(* CODESYS project tc2_mc2.library
   Company: Beckhoff Automation GmbH
   DefaultNamespace: Tc2_MC2
   Version: 3.3.54.0
   Placeholder: Tc2_MC2
   Author: Beckhoff Automation GmbH
   Description: TwinCAT Motion Control Library (PlcOpen) v2.0
   Title: Tc2_MC2

Project tree, tasks and I/O mapping:
  libraries: Tc2_Math, * (Beckhoff Automation GmbH); Tc2_Standard, * (Beckhoff Automation GmbH); Tc2_System, * (Beckhoff Automation GmbH); Tc3_Module, * (Beckhoff Automation GmbH)
  Data types/
    [Internal]/
      DriveOperationMode/
        data type _ST_TcNC_ReadDriveOperationModeRequest
        data type _ST_TcNC_ReadDriveOperationModeResponse
        data type _ST_TcNC_WriteDriveOperationMode
      TcNC/
        ADS Axis/
          data type _ST_NCADS_Axis
          data type _ST_NCADS_AxisFunctions
          data type _ST_NCADS_AxisParameter
          data type _ST_NCADS_AxisState
          data type _ST_NCADS_IDXOFFS_AxisFunctions
          data type _ST_NCADS_IDXOFFS_AxisParameter
          data type _ST_NCADS_IDXOFFS_AxisState
        ADS Table/
          data type _ST_NCADS_IDXOFFS_TableFunctions
          data type _ST_NCADS_IDXOFFS_TableParameter
          data type _ST_NCADS_Table
          data type _ST_NCADS_TableFunctions
          data type _ST_NCADS_TableParameter
        data type _E_TcNC_CmdState
        data type _E_TcNC_CmdTypeNewTargPosAndVelo
        data type _E_TcNC_PosSetType
        data type _E_TcNC_ServoState
        data type _E_TcNC_SlaveTypes
        data type _E_TcNC_StartPosType
        data type _E_TcNC_TargPosType
        data type _ST_TcNC_Compensation2
        data type _ST_TcNC_CoupleSlave
        data type _ST_TcNC_CoupleSlaveMultiMaster
        data type _ST_TcNC_CoupleSlaveMultiMaster2
        data type _ST_TcNC_DecoupleSlave
        data type _ST_TcNc_OperationModes
        data type _ST_TcNC_PhasingRequest
        data type _ST_TcNC_SetEncoderSaclingFactor
        data type _ST_TcNC_SetPos
        data type _ST_TcNC_SetPosOnTheFly
        data type _ST_TcNc_SinusMotion
        data type _ST_TcNC_StopInfoRequest
        data type _ST_TcNC_StopInfoResponse
        data type _ST_TcNc_TouchProbeActivation
        data type _ST_TcNc_TouchProbeDeactivation
        data type _ST_TcNc_TouchProbeStatusRequest
        data type _ST_TcNc_TouchProbeStatusResponse
        data type _ST_TcNC_UniversalAxisTorqueStartRequest
        data type _ST_TcNC_UnversalAxisStartRequest
        data type _ST_TcNC_UnversalAxisStartResponse
      data type _E_ParameterType
      data type _E_PhasingState
      data type _E_ReadWriteParameterMode
      data type _E_SinusMotionMode
      data type _E_TcMC_STATES
      data type _E_TouchProbeState
      data type _InternalAxisRefData
      data type _ST_FunctionBlockResults
      data type _ST_NcIoOutputData
      data type _ST_ParaStruct
    Axis Reference/
      function block AXIS_REF [ST]: ReadStatus
      data type ST_AdsAddress
    BacklashCompensation/
      data type ST_BacklashCompensationOptions
    DriveOperationMode/
      data type E_DriveOperationMode
      data type ST_DriveOperationModeOptions
    Gearing/
      data type E_GearInMultiMasterSyncMode
      data type ST_GearInDynOptions
      data type ST_GearInMultiMasterOptions
      data type ST_GearInOptions
      data type ST_GearOutOptions
    Homing/
      data type E_EncoderReferenceMode
      data type MC_HomingMode
      data type ST_HomingOptions
    Motion/
      data type E_JogMode
      data type E_PositionType
      data type MC_BufferMode
      data type MC_Direction
      data type ST_MoveOptions
    Nc Process Data/
      data type E_NcIoDevice
      data type E_NcIoOutput
    Phasing/
      data type E_PhasingType
      data type ST_PhasingOptions
    Position Correction/
      data type E_AxisPositionCorrectionMode
      data type ST_PositionCompensationOptions
      data type ST_PositionCompensationTableElement
      data type ST_PositionCompensationTableParameter
    SelectControlLoop/
      data type E_SelectControlLoopType
      data type ST_SelectControlLoop
    Status and Parameter/
      data type E_AxisErrorCodes
      data type E_DisableMode
      data type E_NcAxisType
      data type E_NcDriveType
      data type E_NcEncoderType
      data type E_ReadMode
      data type E_SetScalingFactorMode
      data type E_WorkDirection
      data type MC_AxisParameter
      data type MC_AxisStates
      data type ST_AxisComponents
      data type ST_AxisOpModes
      data type ST_AxisParameterSet
      data type ST_AxisStatus
      data type ST_DriveAddress
      data type ST_McOutputs
      data type ST_NcApplicationRequest
      data type ST_PowerOptions
      data type ST_SetEncoderScalingOptions
      data type ST_SetPositionOptions
      data type ST_TableCharacValues
    Stepper/
      data type E_DestallDetectMode
      data type E_DestallMode
      data type ST_PowerStepperStruct
    Superposition/
      data type E_SuperpositionAbortOption
      data type E_SuperpositionMode
      data type ST_SuperpositionOptions
    Torque Control/
      data type ST_TorqueControlOptions
    Touch Probe/
      data type E_SignalEdge
      data type E_SignalSource
      data type E_TouchProbe
      data type E_TouchProbeMode
      data type MC_TouchProbeRecordedData
      data type TRIGGER_REF
  Global Variables/
    global variables Global_Variables
  POUs/
    [Internal]/
      ADS/
        function block _TcMC_ADSRDWRT [ST]
        function block _TcMC_ADSREAD [ST]
        function block _TcMC_ADSWRITE [ST]
      Axis Status Flag Functions/
        function F_AxisCamDataQueued [ST]
        function F_AxisCamScalingPending [ST]
        function F_AxisCamTableQueued [ST]
        function F_AxisControlLoopClosed [ST]
        function F_AxisDriveLimitActive [ST]
        function F_AxisExternalLatchValid [ST]
        function F_AxisGotNewTargetPosition [ST]
        function F_AxisHasBeenStopped [ST]
        function F_AxisHasExtSetPointGen [ST]
        function F_AxisHasJob [ST]
        function F_AxisInErrorState [ST]
        function F_AxisInPositionWindow [ST]
        function F_AxisInProtectedMode [ST]
        function F_AxisInPTPmode [ST]
        function F_AxisIoDataIsInvalid [ST]
        function F_AxisIsAtTargetPosition [ST]
        function F_AxisIsCalibrated [ST]
        function F_AxisIsCalibrating [ST]
        function F_AxisIsCompensating [ST]
        function F_AxisIsCoupled [FBD]
        function F_AxisIsMoving [ST]
        function F_AxisIsMovingBackwards [ST]
        function F_AxisIsMovingEndless [ST]
        function F_AxisIsMovingForward [ST]
        function F_AxisIsNotMoving [ST]
        function F_AxisIsReady [ST]
        function F_AxisJobPending [ST]
        function F_AxisMotionCommandsLocked [ST]
        function F_AxisPhasingActive [ST]
        function F_AxisReachedConstantVelocity [ST]
      Beta Function Blocks/
        Position Correction/
          function block MC_TableBasedPositionCompensation [ST]
        Sinus motion/
          function block MC_SinusOscillation [ST]
          function block MC_SinusSequence [ST]
        function block MC_ReadApplicationRequest [ST]
        function block MC_ReadStopInfo [ST]
      Objects/
        data type _FBAXIS_REF
        function block _TCMCGLOBAL [ST]: ReadDeviceInfo
      function _F_AxisState [ST]
      function _F_GetIndexGroup [ST]
      function _F_GetTcAxisObjectId [ST]
      function _F_GetTcDriveObjectId [ST]
      function _F_GetTcEncoderObjectId [ST]
      function _F_Init [ST]
      function _F_NcCycleCounterUpdated [ST]
      function _F_NcNoOfCycleCounterUpdated [ST]
      function _F_ReadStatus [ST]
      function _F_TcMC_DWORD_TO_HEXSTR [ST]
      function _F_TcMC_DWORD_TO_HEXSTR2 [ST]
      function _F_TcMC_IsValidAxisRef [ST]
      function _F_TcMC_IsValidRef [ST]
      function _F_TcMC_Round [ST]
      function _F_UpdateNcCycleCounter [ST]
      function block _FB_MoveSinusGeneric [ST]
      function block _FB_MoveUniversalGeneric [ST]: ActCalcDiffCmdNo, ActErrorMessage, ActMonitorAbortTorque, ActMonitorContinousMotion, ActMonitorContinuousTorque, ActMonitorDiscreteMotion, ActMonitorStop, ActNcCycleCounter
      function block _FB_PhasingGeneric [ST]
      function block _FB_PositionCorrectionTableLookup [ST]: ActIsCompensationDirection
      function block _FB_ReadWriteParameter [ST]
      function block _FB_WriteParameterPersistent [ST]
    [obsolete]/
      function F_GetVersion_TcMC2 [ST]
    Administrative/
      Axis Functions/
        function block MC_Power [ST]
        function block MC_Reset [ST]
        function block MC_SetPosition [ST]
      Extensions/
        DriveOperationMode/
          function block MC_ReadDriveOperationMode [ST]
          function block MC_WriteDriveOperationMode [ST]
        function block MC_BacklashCompensation [ST]
        function block MC_CalcDynamicsByRampTime [ST]
        function block MC_OverrideFilter [ST]
        function block MC_PositionCorrectionLimiter [ST]
        function block MC_PowerStepper [ST]
        function block MC_ReadDriveAddress [ST]
        function block MC_SelectControlLoop [ST]
        function MC_SetAcceptBlockedDriveSignal [ST]
        function block MC_SetEncoderScalingFactor [ST]
        function block MC_SetOverride [ST]
        function block MC_WriteNcIoOutput [ST]
      External Set Point Generator/
        function block MC_ExtSetPointGenDisable [ST]
        function block MC_ExtSetPointGenEnable [ST]
        function MC_ExtSetPointGenFeed [ST]
      Status and Parameter/
        function block MC_ReadActualPosition [ST]
        function block MC_ReadActualVelocity [ST]
        function block MC_ReadAxisComponents [ST]
        function block MC_ReadAxisError [ST]
        function block MC_ReadBoolParameter [ST]
        function block MC_ReadLargeParameter [ST]
        function block MC_ReadParameter [ST]
        function block MC_ReadParameterSet [ST]: ActGetSizeOfParameterSet
        function block MC_ReadStatus [ST]
        function block MC_WriteBoolParameter [ST]
        function block MC_WriteBoolParameterPersistent [ST]
        function block MC_WriteLargeParameter [ST]
        function block MC_WriteLargeParameterPersistent [ST]
        function block MC_WriteParameter [ST]
        function block MC_WriteParameterPersistent [ST]
      Touch Probe/
        function block MC_AbortTrigger [ST]
        function block MC_TouchProbe [ST]: ActTouchProbeActivate, ActTouchProbeMonitorActivity, ActTouchProbeMonitoring, ActTouchProbeMonitorLatchValid, ActTouchProbeMonitorPlcEvent, ActTouchProbeStartupInit
    Motion/
      Gearing/
        function block MC_GearIn [ST]: ActGearInDyn, WriteGearRatio
        function block MC_GearInDyn [ST]
        function block MC_GearInMultiMaster [ST]: ActGearInMultiMasterV1, ActGearInMultiMasterV2
        function block MC_GearOut [ST]
      Homing/
        function block MC_Home [ST]
      Manual Motion/
        function block MC_Jog [ST]: ActCheckJogEnd, ActJogMove
      Phasing/
        function block MC_HaltPhasing [FBD]
        function block MC_PhasingAbsolute [FBD]
        function block MC_PhasingRelative [FBD]
      Point To Point Motion/
        function block MC_Halt [FBD]
        function block MC_MoveAbsolute [FBD]
        function block MC_MoveAdditive [FBD]
        function block MC_MoveContinuousAbsolute [FBD]
        function block MC_MoveContinuousRelative [FBD]
        function block MC_MoveModulo [ST]: MC_MoveModuloCall
        function block MC_MoveRelative [FBD]
        function block MC_MoveVelocity [FBD]
        function block MC_Stop [ST]: ActStop
      Superposition/
        function block MC_AbortSuperposition [ST]
        function block MC_MoveSuperImposed [ST]
      Torque Control/
        function block MC_AbortTorqueControl [FBD]
        function block MC_TorqueControl [FBD]
  Version/
    global variables Global_Version
*)

// Data types/[Internal]/DriveOperationMode/_ST_TcNC_ReadDriveOperationModeRequest
{attribute 'conditionalshow'}
TYPE _ST_TcNC_ReadDriveOperationModeRequest :
STRUCT
	nReserved1 : UDINT;	// RESERVED1 (e.g. 'ULONG nCtrlLoopIndex')
	nReserved2 : UDINT;	// TC3 specific (natural alignment)
END_STRUCT
END_TYPE

// Data types/[Internal]/DriveOperationMode/_ST_TcNC_ReadDriveOperationModeResponse
{attribute 'conditionalshow'}
TYPE _ST_TcNC_ReadDriveOperationModeResponse :
STRUCT
	eTcNc3DrvOpMode : E_DriveOperationMode;	// >=0 [1] actual drive operation mode (enum NC3 Drive Operation Modes) (NC data type equal to ULONG)
    nReserved		: UDINT;	// RESERVED (e.g. OTCID    nObjectId, data type OTCID is equal to ULONG)
END_STRUCT
END_TYPE

// Data types/[Internal]/DriveOperationMode/_ST_TcNC_WriteDriveOperationMode
{attribute 'conditionalshow'}
TYPE _ST_TcNC_WriteDriveOperationMode :
STRUCT
	eTcNc3DrvOpMode : E_DriveOperationMode;	// enum NC3 Drive Operation Modes (signed value)(NC data type equal to ULONG)
	nReserved0 : UDINT;	// RESERVED1 (e.g. ULONG nCtrlLoopIdx [0;1,2,...])
	nReserved1 : UDINT; // RESERVED2 (e.g. 'OTCID nObjectId', data type equal to ULONG) (ObjId 0x0 is invalid, ObjID 0xFFFFFFFF is a joker (always allowed))
	nReserved2 : UDINT; // RESERVED3 
END_STRUCT
END_TYPE

// Data types/[Internal]/TcNC/ADS Axis/_ST_NCADS_Axis
{attribute 'conditionalshow'}
TYPE _ST_NCADS_Axis :
STRUCT
	Parameter	:	_ST_NCADS_AxisParameter;
	State		:	_ST_NCADS_AxisState;
	Functions	:	_ST_NCADS_AxisFunctions;
END_STRUCT
END_TYPE

// Data types/[Internal]/TcNC/ADS Axis/_ST_NCADS_AxisFunctions
{attribute 'conditionalshow'}
TYPE _ST_NCADS_AxisFunctions :
STRUCT
	IDXGRP		:	UDINT := 16#4200;
	IDXOFFS	:	_ST_NCADS_IDXOFFS_AxisFunctions;
END_STRUCT
END_TYPE

// Data types/[Internal]/TcNC/ADS Axis/_ST_NCADS_AxisParameter
{attribute 'conditionalshow'}
TYPE _ST_NCADS_AxisParameter :
STRUCT
	IDXGRP		:	UDINT := 16#4000;
	IDXOFFS	:	_ST_NCADS_IDXOFFS_AxisParameter;
END_STRUCT
END_TYPE

// Data types/[Internal]/TcNC/ADS Axis/_ST_NCADS_AxisState
{attribute 'conditionalshow'}
TYPE _ST_NCADS_AxisState :
STRUCT
	IDXGRP		:	UDINT := 16#4100;
	IDXOFFS	:	_ST_NCADS_IDXOFFS_AxisState;
END_STRUCT
END_TYPE

// Data types/[Internal]/TcNC/ADS Axis/_ST_NCADS_IDXOFFS_AxisFunctions
{attribute 'conditionalshow'}
TYPE _ST_NCADS_IDXOFFS_AxisFunctions :
STRUCT
	RESET					: UDINT := 16#0001;
	STOP					: UDINT := 16#0002;
	CLEAR					: UDINT := 16#0003;
	EMERGENCYSTOP		: UDINT := 16#0004;
	PARAMETRIZEDSTOP	: UDINT := 16#0005;
	INITIALIZE				: UDINT := 16#0007;	(* Initialize Axis *)
	ORIENTEDSTOP			: UDINT := 16#0009;	(* 19.04.04 issue #2470 *)
	CALIBR					: UDINT := 16#0010;
	NEWTARGPOS			: UDINT := 16#0011;
	NEWTARGPOSANDVELO	: UDINT := 16#0012;
	CHANGEDYNAMICPARAM	: UDINT := 16#0015;	(* NEU: Neue Dynamikparameter (Acc;Dec) fuer Positionierung *)
	UNIVERSALSTART		: UDINT := 16#0016;	(* 05.03.07: new 'axis start and restart' command with buffer mode (issue #2786+#3276) *)
	SLAVEUNIVERSALSTART	: UDINT := 16#0017;	(* 24.02.09: decoupling command with succeding universal axis start commanded to a slave axis *)
	RELEASEAXISLOCK			: UDINT := 16#0018; (* 10.12.18 release axis lock for motion commands *)
(*	ONLINESTART			: UDINT := 16#0017;*)	(* 05.03.07: new 'axis start and restart' command (online start) (issue #2786+#3276) *)
	SETEXTERNALERROR	: UDINT := 16#0019;	(* 06.10.04: Externen Achsfehler setzen (Laufzeitfehler) issue #2665 *)
	SETPOS					: UDINT := 16#001A;
	SETCALFLAG			: UDINT := 16#001B;	(* "ist referenziert"-Flag setzen *)
	SETACTPOS				: UDINT := 16#001C;	(* nur Istwertsetzen ohne Sollwertaenderung !!! *)
	SETDRIVEPOS			: UDINT := 16#001D;	(* antriebsseitiges Istwertsetzen *)
	SETENCODERSCALING	: UDINT := 16#001E;	(* 17.07.08: "Fliegende Änderung des Skalierungsfaktors" *)
	SETPOSONTHEFLY		: UDINT := 16#001F;	(* 29.11.05: "Fliegendes Istwert Setzen" (betrifft Ist - und Sollwert) (issue #3017) *)
	START					: UDINT := 16#0020;
	STARTEXT				: UDINT := 16#0021;
	STARTVELOCHANGE		: UDINT := 16#0022;	(* special function for MMW *)
	ENABLEEXTGEN			: UDINT := 16#0023;	(* enable/start external setpoint values *)
	DISABLEEXTGEN			: UDINT := 16#0024;	(* disable/stop external setpoint values *)
	REVERSINGSEQUENCE	: UDINT := 16#0025;
	STARTDRVOUT			: UDINT := 16#0026;
	STOPDRVOUT			: UDINT := 16#0027;
	CHANGEDRVOUT		: UDINT := 16#0028;
	JUMPTOOVERRIDE		: UDINT := 16#0029;	(* 04.11.04: jump to actual override value and froze them until change (issue #2697) *)
(*	SETABSOLUTEMEASURING: UDINT := 16#002A;	removed 20091106 KSt *)	(* 29.11.05: "Fliegendes Istwert Setzen" (betrifft Ist - und Sollwert) (issue #3017) *)
	EXTSETGENUNIVERSALSTART	: UDINT := 16#002B;	(* 23.11.10: deactivation of external setpoint generator with succeding universal axis start command *)
	UNIVERSALTORQUESTART	: UDINT := 16#002D;	(* 20181210 Fap -  new 'axis torque control start and restart' command with buffer mode *)
	STARTSCOM			: UDINT := 16#0030;	(* start superposition (position compensation) - 21.12.04: nun auch als 'ReadWrite'-Kommando *)
	STOPSCOM				: UDINT := 16#0031;	(* stop superposition (position compensation) *)
	PHASINGREQEUST		: UDINT := 16#0034;	(* start/stop the additional phasing set point generator used for a master/slave phase shift *)
	CPL						: UDINT := 16#0040;	(* Achse koppeln *)
	DECPL					: UDINT := 16#0041;	(* Achse entkoppeln (und optional neue Endposition mit neuer Geschwindigkeit) *)
	CPLCHANGE				: UDINT := 16#0042;	(* Achse Koppelparams ändern *)
	TABCPLCHANGE			: UDINT := 16#0043;	(* 3x TabSlaveAxe Tabelle-Koppelparams ändern *)
	STOPSLAVE				: UDINT := 16#0044;	(* Slave-Stop (Diagonal-Slave / Flying Saw) *)
	CPLTAB					: UDINT := 16#0045;	(* TabSlaveAxe Koppelparams setzen *)
	TABSLVACTIVCOR		: UDINT := 16#0046;	(* 2x TabSlaveAxe Korrekturtabelle aktivieren (mit/ohne Aktivierungsposition) *)
	TABSLVLEAVECYC		: UDINT := 16#0047;	(* TabSlaveAxe	Monozyklische Tabelle beenden *)
	TABSLVCOROFFSET		: UDINT := 16#0048;	(* TabSlaveAxe	Letzter Korrektur Offset *)
	TABSLVSCALING			: UDINT := 16#0049;	(* NEU: Slave-Skalierung der Solo-Tabellenkopplung setzen *)
	CPLSOLOTAB			: UDINT := 16#004A;	(* Solo Tabellen Kopplung *)
	CPLSYNCHRONIZING		: UDINT := 16#004B;	(* Slave Synchronizing Generator ('GearInPos' and 'GearInVelo') *)
	CAMSCALING			: UDINT := 16#004D;	(* Slave Change CAM Scaling (Aenderung der Tabellenskalierung) (issue #2514) *)
	DISABLE				: UDINT := 16#0050;	(* Achse sperren *)
	ENABLE					: UDINT := 16#0051;	(* Achse reaktivieren *)
	CHANGEAXISCTRLLOOP	: UDINT := 16#0052;	(* NEU: Aenderung des aktiven Achsregelkreises *)
	DRIVEDISABLE			: UDINT := 16#0060;	(* Drive-Output der Achse sperren *)
	DRIVEENABLE			: UDINT := 16#0061;	(* Drive-Output der Achse reaktivieren *)
	RELEASEBRAKE			: UDINT := 16#0062;	(* Feststellbremse loesen (Eil/Schleich-Gruppe) *)
	RECONFIGURATE		: UDINT := 16#0070;	(* Achse zurueckfuehren in eigene PTP-Gruppe *)
END_STRUCT
END_TYPE

// Data types/[Internal]/TcNC/ADS Axis/_ST_NCADS_IDXOFFS_AxisParameter
{attribute 'conditionalshow'}
TYPE _ST_NCADS_IDXOFFS_AxisParameter :
STRUCT
	(* NC ADS Index Offsets for Axis Parameters *)
	PARAMSTRUCT				: UDINT := 16#0000;
	ID							: UDINT := 16#0001;
	NAME						: UDINT := 16#0002;
	AXISTYPE					: UDINT := 16#0003;
	CYCLETIME					: UDINT := 16#0004;
	UNITNAME					: UDINT := 16#0005;
	VELOREFSEARCH			: UDINT := 16#0006;
	VELOSYNCSEARCH			: UDINT := 16#0007;
	VELOSLOWMANUAL			: UDINT := 16#0008;
	VELOFASTMANUAL			: UDINT := 16#0009;
	VELOFAST					: UDINT := 16#000A;
	POSAREAENABLE			: UDINT := 16#000F;
	POSAREARANGE			: UDINT := 16#0010;
	MOTCNTRLENABLE			: UDINT := 16#0011;
	MOTCNTRLTIME				: UDINT := 16#0012;
	LOOPENABLE				: UDINT := 16#0013;
	LOOPDISTANCE				: UDINT := 16#0014;
	TARGETPOSENA			: UDINT := 16#0015;
	TARGETPOSRANGE			: UDINT := 16#0016;
	TARGETPOSTIME			: UDINT := 16#0017;
	PULSDISTPOS				: UDINT := 16#0018;
	PULSDISTNEG				: UDINT := 16#0019;
	FADINGACCELERATION		: UDINT := 16#001D;
	FASTAXISSTOPSIGNALTYPE	: UDINT := 16#001E;
	UNITFLAGS					: UDINT := 16#0026;
	VELOMAXIMUM				: UDINT := 16#0027;
	MOTCNTRLRANGE			: UDINT := 16#0028;
	PEHCONTROLENA			: UDINT := 16#0029;
	PEHCONTROLTIME			: UDINT := 16#002A;
	BACKLASHCOMPENA			: UDINT := 16#002B;
	BACKLASH					: UDINT := 16#002C;
	DATAPERSISTENCE			: UDINT := 16#0030;
	HWAMSADDR				: UDINT := 16#0031;
	HWCHNNO					: UDINT := 16#0032;
	APPLICATIONREQUEST 		: UDINT := 16#0033;
	ACC							: UDINT := 16#0101;
	DEC						: UDINT := 16#0102;
	JERK						: UDINT := 16#0103;
	DELAY						: UDINT := 16#0104;
	OVERRIDETYPE				: UDINT := 16#0105;
	VELOJUMPFACTOR			: UDINT := 16#0106;
	REDUCTIONFEEDBACK		: UDINT := 16#0107;
	TOLERANCEBALLAUXAXIS	: UDINT := 16#0108;
	MAXPOSDEVIATIONAUXAXIS 	: UDINT := 16#0109;
	FASTACC					: UDINT := 16#010A;
	FASTDEC					: UDINT := 16#010B;
	FASTJERK					: UDINT := 16#010C;
	REF_POS						: UDINT := 16#0001_0103;
	ENCSEARCHDIR				: UDINT := 16#0001_0101;
	ENCSYNCDIR					: UDINT := 16#0001_0102;
	ENCREFMODE					: UDINT := 16#0001_0107;

(*
	SCALE						= TCNC_IDXOFFS_AXmappedENC | 0x00000006;	// 0x00010006;
	ENABLESOFTENDMIN		= TCNC_IDXOFFS_AXmappedENC | 0x0000000B;	// 0x0001000B;
	ENABLESOFTENDMAX		= TCNC_IDXOFFS_AXmappedENC | 0x0000000C;	// 0x0001000C;
	SOFTENDMIN				= TCNC_IDXOFFS_AXmappedENC | 0x0000000D;	// 0x0001000D;
	SOFTENDMAX				= TCNC_IDXOFFS_AXmappedENC | 0x0000000E;	// 0x0001000E;
	ENABLEPOSDIFF				= TCNC_IDXOFFS_AXmappedCTR | 0x00000010;	// 0x00020010;
	POSDIFFMAX				= TCNC_IDXOFFS_AXmappedCTR | 0x00000012;	// 0x00020012;
	GAINPOS					= TCNC_IDXOFFS_AXmappedCTR | 0x00000102;	// 0x00020102;
	VELOREF					= TCNC_IDXOFFS_AXmappedDRV | 0x00000101;	// 0x00030101;
*)
END_STRUCT
END_TYPE

// Data types/[Internal]/TcNC/ADS Axis/_ST_NCADS_IDXOFFS_AxisState
{attribute 'conditionalshow'}
TYPE _ST_NCADS_IDXOFFS_AxisState :
STRUCT
	ONLINESTRUCT					: UDINT := 16#0000;
	ERROR							: UDINT := 16#0001;
(*
	ACTPOS							= TCNC_IDXOFFS_AXmappedENC | 0x00000002;	// 0x00010002;
	ACTVELO						= TCNC_IDXOFFS_AXmappedENC | 0x00000005;	// 0x00010005;
	ACTACC							= TCNC_IDXOFFS_AXmappedENC | 0x00000006;	// 0x00010006;
	MODULOACTPOS				= TCNC_IDXOFFS_AXmappedENC | 0x00000003;	// 0x00010003;
	MODULOACTTURNS				= TCNC_IDXOFFS_AXmappedENC | 0x00000004;	// 0x00010004;
	ACTINCREMENTS				= TCNC_IDXOFFS_AXmappedENC | 0x00000007;	// 0x00010007;
*)
	SETTASKCYCLE					: UDINT := 16#0009;
	SETPOS							: UDINT := 16#000A;
	SETVELO						: UDINT := 16#000E;
	SETACC							: UDINT := 16#000F;
	MODULOSETPOS				: UDINT := 16#000B;
	MODULOSETTURNS				: UDINT := 16#000C;
	SETDIR							: UDINT := 16#000D;
	TARGETPOSITION				: UDINT := 16#0013;
	REMAININGTIMEANDPOS			: UDINT := 16#0014;
	STOPINFORMATION				: UDINT := 16#0018;
	SETTASKCYCLE_WITHOUTCORR	: UDINT := 16#0019;
	SETPOS_WITHOUTCORR			: UDINT := 16#001A;
	SETVELO_WITHOUTCORR		: UDINT := 16#001E;
	SETACC_WITHOUTCORR			: UDINT := 16#001F;
	SETDIR_WITHOUTCORR			: UDINT := 16#001D;
	COUPLESTATE					: UDINT := 16#0020;
	CPLPARAMS						: UDINT := 16#0022;
	CPLFACTOR						: UDINT := 16#0023;
	AXISCTRLLOOPIDX				: UDINT := 16#0024;
	AXISSETPOINTGENIDX			: UDINT := 16#0025;
	CPLCHARACVALUES				: UDINT := 16#0026;
	CAMINFO						: UDINT := 16#0027;
	CAMSTATUS					: UDINT := 16#0028;	(* activation status etc. *)
(*
	POSDIFF						= TCNC_IDXOFFS_AXmappedCTR | 0x0000000F;	// 0x0002000F;
*)
END_STRUCT
END_TYPE

// Data types/[Internal]/TcNC/ADS Table/_ST_NCADS_IDXOFFS_TableFunctions
{attribute 'conditionalshow'}
TYPE _ST_NCADS_IDXOFFS_TableFunctions :
STRUCT
	(* Index Offset definitions of table functions *)
	CREATETAB				: UDINT := 	16#0001_0000;		(* create table*)
	CREATEMOTIONTAB 		: UDINT := 	16#0001_0010;		(* create motion function table*)
	DELETETAB 				: UDINT := 	16#0002_0000; 		(* delete tables *)
END_STRUCT
END_TYPE

// Data types/[Internal]/TcNC/ADS Table/_ST_NCADS_IDXOFFS_TableParameter
{attribute 'conditionalshow'}
TYPE _ST_NCADS_IDXOFFS_TableParameter :
STRUCT
	MFREADCHARACVALUES	: UDINT := 	16#0000_0050;		(* read characteristic values of a motion function *)
	WRITETABROWS 		: UDINT := 	16#0100_0000;		(* write table *)
(*	WRITETABCOLS 			: UDINT := 	16#0200_0000;	*)	(* write table *)
	WRITEMFTABROWS 		: UDINT := 	16#0500_0000;		(* write motion function table *)
(*	WRITEMFTABCOLS 		: UDINT := 	16#0600_0000;	*)	(* write motion function table *)
(*	READSLAVEPOS 		: UDINT := 	16#0000_0021;	*)	(* read slave table position related to a master position *)
	MFREADTAB 			: UDINT := 	16#0000_0022;		(* read motion function as data table *)
	READSLAVEDYNAMICS 	: UDINT := 	16#0000_0023;		(* read slave table position, velocity and acceleration related to a master position *)
	READMASTERPOSITION 	: UDINT := 	16#0000_0024;		(* read master table position related  to slave position *)
END_STRUCT
END_TYPE

// Data types/[Internal]/TcNC/ADS Table/_ST_NCADS_Table
{attribute 'conditionalshow'}
TYPE _ST_NCADS_Table :
STRUCT
	Parameter	:	_ST_NCADS_TableParameter;
	Functions	:	_ST_NCADS_TableFunctions;
END_STRUCT
END_TYPE

// Data types/[Internal]/TcNC/ADS Table/_ST_NCADS_TableFunctions
{attribute 'conditionalshow'}
TYPE _ST_NCADS_TableFunctions :
STRUCT
	IDXGRP		:	UDINT := 16#A200;
	IDXOFFS	:	_ST_NCADS_IDXOFFS_TableFunctions;
END_STRUCT
END_TYPE

// Data types/[Internal]/TcNC/ADS Table/_ST_NCADS_TableParameter
{attribute 'conditionalshow'}
TYPE _ST_NCADS_TableParameter :
STRUCT
	IDXGRP		:	UDINT := 16#A000;
	IDXOFFS	:	_ST_NCADS_IDXOFFS_TableParameter;
END_STRUCT
END_TYPE

// Data types/[Internal]/TcNC/_E_TcNC_CmdState
{attribute 'conditionalshow'}
TYPE _E_TcNC_CmdState :
 (
	CMDSTATE_SUCCESSFULLY_EXECUTED				:= 1,	(* bit number *)
	CMDSTATE_ABORTED_WITHOUT_ERROR				:= 2,
	CMDSTATE_ENDED_WITH_ERROR					:= 3,
	CMDSTATE_LASTCMD_SUCCESSFULLY_EXECUTED	:= 8,
	CMDSTATE_LASTCMD_ABORTED_WITHOUT_ERROR	:= 9,
	CMDSTATE_LASTCMD_ENDED_WITH_ERROR			:= 10
 );
END_TYPE

// Data types/[Internal]/TcNC/_E_TcNC_CmdTypeNewTargPosAndVelo
{attribute 'conditionalshow'}
TYPE _E_TcNC_CmdTypeNewTargPosAndVelo :
 (
	TCNC_CHANGE_POS						:=  1,		(*Position (instantan)*)
	TCNC_CHANGE_VELO,							(*Geschwindigkeit (instantan)*)
	TCNC_CHANGE_POSANDVELO,					(*Position und Geschwindigkeit (instantan)*)
	TCNC_CHANGE_POS_AT_SWITCHPOS		:=  9,		(*Position (Umschaltposition)*)
	TCNC_CHANGE_VELO_AT_SWITCHPOS,			(*Geschwindigkeit (Umschaltposition)*)
	TCNC_CHANGE_POSANDVELO_AT_SWITCHPOS,	(*Position und Geschwindigkeit (Umschaltposition)*)
	TCNC_REACH_VELO_AT_POS				:= 14		(*neue Geschwindigkeit wird an einer bestimmten Position erreicht *)
 );
END_TYPE

// Data types/[Internal]/TcNC/_E_TcNC_PosSetType
{attribute 'conditionalshow'}
TYPE _E_TcNC_PosSetType : (* mode is used with MC_SetPosition *)
(
	TCNC_POSSETTYPE_ABSOLUTE		:= 1,	(*Absolute position*)
	TCNC_POSSETTYPE_RELATIVE			(*Relative position*)
) UINT;
END_TYPE

// Data types/[Internal]/TcNC/_E_TcNC_ServoState
{attribute 'conditionalshow'}
TYPE _E_TcNC_ServoState :
 (
	TCNC_INACTIVE 	:= 0,
	TCNC_RUNNING,
	TCNC_OVERRIDE_ZERO,			(* axis is executing a job but override is zero *)
	TCNC_PHASE_VELOCONST,		(* aixs is moving at constant velocity *)
	TCNC_PHASE_ACCPOS,			(* axis is accelerating *)
	TCNC_PHASE_ACCNEG,			(* axis is decelerating *)
	TCNC_PHASE_TORQUECONST,		(* 20181210 Fap - axis is moving at constant torque *)

	(* slaves only *)
	TCNC_PHASE_PREPHASE := 11, 	(* slave axis is in a motion pre-phase - slaves only *)
	TCNC_PHASE_SYNCHRONIZING, 	(* slave axis is synchronizzing slaves only *)
	TCNC_PHASE_SYNCHRONOUS, 	(* slaves only *)

	(* two speed axes only *)
	TCNC_PHASE_TWOSPEED_MOVING := 21,	(* GVGSTATE_TWOSPEED_21 *)

	(* external set point generation - from Tc 2.11 R2 *)
	TCNC_PHASE_EXTSETGEN_MODE1 := 41,	(* external set point generator active *)
	TCNC_PHASE_EXTSETGEN_MODE2		(* internal and external set point generator active *)
 );
END_TYPE

// Data types/[Internal]/TcNC/_E_TcNC_SlaveTypes
{attribute 'conditionalshow'}
TYPE _E_TcNC_SlaveTypes :
(
	TCNC_SLAVETYPE_LINEAR							:=	1,	(* Lineare Kopplung (Geradengleichung) *)
	TCNC_SLAVETYPE_FLYINGSAW_ONVELOCITY		:= 	2,	(* diagonal synchron. Aufkoppeln schnellstens auf Geschwindigkeit *)
	TCNC_SLAVETYPE_FLYINGSAW_ONPOSITION		:=	3,	(* diagonal synchron. Aufkoppeln auf Position und Geschwindigkeit *)
	TCNC_SLAVETYPE_FLYINGSAW_QUADRATIC		:=	4,	(* diagonal synchron. Aufkoppeln (quadratisches Geschw.-Profil) *)
	TCNC_SLAVETYPE_SYNCHRONIZING_ONVELO		:= 	5,	(* synchron. Aufkoppeln instantan auf Geschwindigkeit *)
	TCNC_SLAVETYPE_SYNCHRONIZING_ONPOS       	 	:= 	6,	(* synchron. Aufkoppeln auf Positionen und Geschwindigkeit *)
	TCNC_SLAVETYPE_SYNCJERKSETTER_ONVELO       	:= 	7,	(* synchron. Aufkoppeln auf Geschwindigkeit (zeitbasiert mittels Ruck-Steller) *)
	TCNC_SLAVETYPE_TABULAR						:=	10,	(* Tabellen-Kopplung ("simple/standard tabular slave") *)
	TCNC_SLAVETYPE_MULTITABULAR					:= 	11,	(* Tabellen-Kopplung ("multiscalable multi-tabular slave") *)
	TCNC_SLAVETYPE_FLYINGMODULO_LINEAR			:=	12,	(* Modulo Kopplung auf Position und/oder Geschwindigkeit mit anschliessender Linear Kopplung ("Schuette") *)
	TCNC_SLAVETYPE_MOTIONFUNCTIONTABULAR		:=	13,	(* Tabellen-Kopplung "motion functions" *)
	TCNC_SLAVETYPE_UNIVERSALTABULAR			:=	14,	(* Tabellen-Kopplung, universal tabular type substitues TABULAR, MULTITABULAR and MOTIONFUNCTION - 08.07.05 *)
	TCNC_SLAVETYPE_LINEAR_CYCLICCHANGES_RAMP	:=	15,	(* Lineare Kopplung (Geradengleichung) mit zyklischer Koppelfaktoraenderung *)
	TCNC_SLAVETYPE_BILINEAR						:=	16,	(* 27.04.01: Zweifach Lineare Kopplung (Geradengleichung)*)
	TCNC_SLAVETYPE_LINEAR_MULTIMASTER		:=	17,	(* 29.05.08: Lineare Multi-Master-Kopplung ('MC_GearInMultiMaster') *)
	TCNC_SLAVETYPE_CONST_SURFACEVELO_RAMP	:=	18	(* Verrechnete Winkelgeschwindigkeit fuer konstante Oberflaechengeschwindig. in Abhaengigkeit vom Radiusistwert des Enc.2 *)
);
END_TYPE

// Data types/[Internal]/TcNC/_E_TcNC_StartPosType
{attribute 'conditionalshow'}
TYPE _E_TcNC_StartPosType :
(
	TCNC_START_ABSOLUTE					:= 1,		(*Start to absolute position*)
	TCNC_START_RELATIVE					:= 2,		(*Start to relative position*)
	TCNC_START_ENDLESS_PLUS				:= 3,		(*Start to endless positive position*)
	TCNC_START_ENDLESS_MINUS			:= 4,		(*Start to endless negative position*)
	TCNC_START_MODULO					:= 5,		(*Start to modulo position *)
	TCNC_START_ADDITIVE					:= 6,		(*Start to a position relative to the last recent target position *)
	TCNC_START_MODULO_SHORT				:= 261, 	(*Start to modulo position *)
 	TCNC_START_MODULO_PLUS				:= 517, 	(*Start to modulo position *)
 	TCNC_START_MODULO_MINUS				:= 773, 	(*Start to modulo position *)
	TCNC_START_MODULO_CURRENT			:= 1029,	(* start to modulo position in current direction *)
 	TCNC_START_ABS_INTERNAL				:= 9, 		(*Start to absolute position, internal use*)
	TCNC_START_ENDLESSPLUS_SLOWMANUAL	:= 272,		(* manual jog mode *)
	TCNC_START_ENDLESSMINUS_SLOWMANUAL	:= 273,		(* manual jog mode *)
	TCNC_START_ENDLESSPLUS_FASTMANUAL	:= 528,		(* manual jog mode *)
	TCNC_START_ENDLESSMINUS_FASTMANUAL	:= 529,		(* manual jog mode *)
	TCNC_START_STOPANDLOCK				:= 4096,	(* stop axis and lock against any motion commands *)
	TCNC_START_HALT						:= 8192,	(* halt axis - can be interrupted by any motion commands *)
	TCNC_START_TORQUE_ABORT				:= 12288,	(* 20181210 Fap - halt torque control *)
	TCNC_START_TORQUE_ABSOLUTE			:= 12289,	(* 20181210 Fap - Start torque control absolute *)
	TCNC_START_TORQUE_RELATIVE			:= 12290	(* 20190108 Fap - Start torque control relative NOT IMPLEMENTED *)
) UINT;
END_TYPE

// Data types/[Internal]/TcNC/_E_TcNC_TargPosType
{attribute 'conditionalshow'}
TYPE _E_TcNC_TargPosType :
(
	TCNC_POS_ABSOLUTE		:= 1,	(*Absolute position*)
	TCNC_POS_RELATIVE,			(*Relative position*)
	TCNC_POS_MODULO			:= 5,	(*Modulo position*)
	TCNC_POS_ABS_INTERNAL	:= 9	(*Absolute position, internal use*)
);
END_TYPE

// Data types/[Internal]/TcNC/_ST_TcNC_Compensation2
{attribute 'conditionalshow'}
TYPE _ST_TcNC_Compensation2 :	(* internal use with MC_MoveSuperimposed_2 *)
STRUCT
	nCompType	:	UDINT;	(* E_SuperpositionMode *)
	nReserved1	:	UDINT;
	fAccPlus		:	LREAL;
	fAccMinus	:	LREAL;
	fVeloDiff		:	LREAL;
	fVeloProcess	:	LREAL;
	fDistance	:	LREAL;	(* distance to compensate *)
	fLength		:	LREAL;	(* distance moved during compensation *)
	nWarningId	: 	UDINT;	(* documented as error code *)
	nReserved2	:	UDINT;
END_STRUCT
END_TYPE

// Data types/[Internal]/TcNC/_ST_TcNC_CoupleSlave
{attribute 'conditionalshow'}
TYPE _ST_TcNC_CoupleSlave :
STRUCT
	nSlaveType		:	UDINT;
	nMasterAxisId	:	UDINT;
	nMasterSubIdx	:	UDINT;
	nSlaveSubIdx		:	UDINT;
	fCoupleParam1	:	LREAL;
	fCoupleParam2	:	LREAL;
	fCoupleParam3	:	LREAL;
	fCoupleParam4	:	LREAL;
END_STRUCT
END_TYPE

// Data types/[Internal]/TcNC/_ST_TcNC_CoupleSlaveMultiMaster
{attribute 'conditionalshow'}
TYPE _ST_TcNC_CoupleSlaveMultiMaster :
STRUCT
	nSlaveType		:	UDINT;
	nMasterAxisId	:	UDINT;
	nMasterSubIdx	:	UDINT;
	nSlaveSubIdx		:	UDINT;
(*	nMasterID1 = nMasterAxisId *)
	nMasterID2		:	UDINT;
	nMasterID3		:	UDINT;
	nMasterID4		:	UDINT;
	nMasterID5		:	UDINT;
	nMasterID6		:	UDINT;
	nMasterID7		:	UDINT;
	nMasterID8		:	UDINT;
	nReserved1		:	UDINT;
	fSlaveAcceleration:	LREAL;
	nCheckAndOpMode:	DWORD;
	nReserved2		:	UDINT;
END_STRUCT
END_TYPE

// Data types/[Internal]/TcNC/_ST_TcNC_CoupleSlaveMultiMaster2
{attribute 'conditionalshow'}
TYPE _ST_TcNC_CoupleSlaveMultiMaster2 :
STRUCT
	nSlaveType		:	UDINT;
	nMasterAxisId	:	UDINT;
	nMasterSubIdx	:	UDINT;
	nSlaveSubIdx		:	UDINT;
(*	nMasterID1 = nMasterAxisId *)
	nMasterID2		:	UDINT;
	nMasterID3		:	UDINT;
	nMasterID4		:	UDINT;
	nMasterID5		:	UDINT;
	nMasterID6		:	UDINT;
	nMasterID7		:	UDINT;
	nMasterID8		:	UDINT;
	nReserved1		:	UDINT;
	fSlaveMaxAcc	:	LREAL;
	nCheckAndOpMode : 	DWORD;
	nReserved2		:	UDINT;
(*	// Erweiterungen fuer NEW VERSION V2 *)
	fSlaveMaxDec	:	LREAL;
	fSlaveMaxJerk	:	LREAL;
	fSlaveMaxVelo	:	LREAL;
	fReserved3		:	LREAL;
	fReserved4		:	LREAL;
END_STRUCT
END_TYPE
(* 	nCheckAndOpMode is a 32 bit array
Bits:
 0:	VelocitySynchronizationOnly		
 1:	
 2:
*)

// Data types/[Internal]/TcNC/_ST_TcNC_DecoupleSlave
{attribute 'conditionalshow'}
TYPE _ST_TcNC_DecoupleSlave :
STRUCT
	nDecoupleMode	:	UDINT;
	nReserved		:	UDINT;
	fNewPosEnd	:	LREAL;
	fNewVeloRequ	:	LREAL;
	fAcceleration	:	LREAL;
	fDeceleration	:	LREAL;
	fJerk			:	LREAL;
END_STRUCT
END_TYPE

// Data types/[Internal]/TcNC/_ST_TcNc_OperationModes
{attribute 'conditionalshow'}
TYPE _ST_TcNc_OperationModes :
STRUCT
	(* OpModeDWord in cyclic interface *)
(*   0 *)	PosAreaControl	:	DWORD := 2#0000_0000_0000_0000_0000_0000_0000_0001;
(*   1 *)	TargetPosControl	:	DWORD := 2#0000_0000_0000_0000_0000_0000_0000_0010;
(*   2 *)(*	Loop			:	DWORD := 2#0000_0000_0000_0000_0000_0000_0000_0100;*)
(*   3 *)(*	MotionControl		:	DWORD := 2#0000_0000_0000_0000_0000_0000_0000_1000;*)
(*   4 *)(*	PEHTimeControl	:	DWORD := 2#0000_0000_0000_0000_0000_0000_0001_0000;*)
(*   5 *)(*	BacklashComp	:	DWORD := 2#0000_0000_0000_0000_0000_0000_0010_0000;*)
(*   6 *)(*	DelayedErrorReaction *)
(*   7 *)(*	Modulo *)
(*   8 *)(*	SimulationAxis *)
	(* bits 9 .. 11 reserved for supplement products *)
(*   12 *)	StopMonitoring 	:	DWORD := 2#0000_0000_0000_0000_0001_0000_0000_0000;
	(* bits 13 .. 15 reserved *)
(* 16 *)(*	PosDiffControl  	:	DWORD := 2#0000_0000_0000_0001_0000_0000_0000_0000;*)
(* 17 *)(*	VeloDiffControl	:	DWORD := 2#0000_0000_0000_0010_0000_0000_0000_0000;*)
(* 18 *)(*	SoftEndMinControl	:	DWORD := 2#0000_0000_0000_0100_0000_0000_0000_0000;*)
(* 19 *)(*	SoftEndMaxControl:	DWORD := 2#0000_0000_0000_1000_0000_0000_0000_0000;*)
(* 20 *)(*	ActPosCorrection	:	DWORD := 2#0000_0000_0001_0000_0000_0000_0000_0000;*)
(* 21 *)	AllowSlaveCommands :DWORD	:= 2#0000_0000_0010_0000_0000_0000_0000_0000;
(* 22 *)(*	AllowExtSetGenAxisCommands*)
(* 23 *)(*	ApplicationRequest*)
	(* bits 24 .. 31  *)
(* 24 *)(* 	NcStartTick : BYTE NC cycle counter *)
END_STRUCT
END_TYPE

// Data types/[Internal]/TcNC/_ST_TcNC_PhasingRequest
{attribute 'conditionalshow'}
TYPE _ST_TcNC_PhasingRequest :	(* internal use with MC_MoveSuperimposed_2 (NCADS_STARTPHASING) *)
STRUCT
	nPhasingType	:	UDINT;	(* phasing type absolute or relative *)
	nControlMask		:	UDINT;	(* internal control mask (RESERVED) *)
	nMasterAxisID	: 	UDINT;	(* Optional: master axis ID (for multi cam) *)
	nReserved1		: 	UDINT;

	fPhaseShift		:	LREAL;	(* phasing shift (distance)		[mm] *)
	fVelo			:	LREAL;	(* maximum velocity (> 0)		[mm/s] *)
	fAcc				:	LREAL;	(* maximum acceleration (>= 0)	[mm/s^2] *)
	fDec			:	LREAL;	(* maximum deceleration (>= 0)	[mm/s^2] *)
	fJerk			:	LREAL;	(* maximum jerk (>= 0)			[mm/s^3] *)

	fReserved		: 	ARRAY[2..5] OF LREAL;

	nReserved6		: 	UDINT;
	nBufferMode		: 	UDINT;	(* NOT USED YET: 'buffer mode' *)
	fBlendingPos		:	LREAL;	(* NOT USED YET: optional blending position *)
END_STRUCT
END_TYPE

// Data types/[Internal]/TcNC/_ST_TcNC_SetEncoderSaclingFactor
{attribute 'conditionalshow'}
TYPE _ST_TcNC_SetEncoderSaclingFactor :
STRUCT
 	nEncoderScalingFactorType	:	UINT;
	nCtrlWord					:	UINT; 	(* additional option flags *)	(* added KSt 2009-04-09 *)
	nReserved					:	UDINT;
	fEncoderScalingFactor		:	LREAL;
END_STRUCT
END_TYPE

// Data types/[Internal]/TcNC/_ST_TcNC_SetPos
{attribute 'conditionalshow'}
TYPE _ST_TcNC_SetPos :
STRUCT
	nPosIstType		:	UDINT;
	nReserved		:	UDINT;
	fNewPosIst		:	LREAL;
	fReserved		:	LREAL;
END_STRUCT
END_TYPE

// Data types/[Internal]/TcNC/_ST_TcNC_SetPosOnTheFly
{attribute 'conditionalshow'}
TYPE _ST_TcNC_SetPosOnTheFly :
STRUCT
	nPosSetType		: 	UDINT; 	(*_E_TcNC_PosSetType *)	(* Absolute, Relative - added KSt 2009-01-28 *)
	nCtrlDWord		:	UDINT; 	(* additional option flags *)	(* added KSt 2009-01-28 *)
 	fPreviousActualPos:	LREAL;	(* value not used any longer since 2009-01-28 *)
	fNewActualPos	:	LREAL;
	nReserved		:	ARRAY[1..2] OF DWORD;	(* added KSt 2009-01-28 *)
END_STRUCT
END_TYPE

// Data types/[Internal]/TcNC/_ST_TcNc_SinusMotion
{attribute 'conditionalshow'}
TYPE _ST_TcNc_SinusMotion :
STRUCT
	StartType 					: UDINT;
	BaseAmplitude 				: LREAL;
	BaseFrequency 				: LREAL;
	StartAmplitudeAtBeginn 		: LREAL;
	FeedConstantMotor 			: LREAL;
	StartFrequency 				: LREAL;
	StopFrequency 				: LREAL;
	StepDuration 				: LREAL;
	NumberMeasurements 			: UDINT;
	NumberParallelMeasurements 	: UDINT;
END_STRUCT
END_TYPE

// Data types/[Internal]/TcNC/_ST_TcNC_StopInfoRequest
{attribute 'conditionalshow'}
TYPE _ST_TcNC_StopInfoRequest :
STRUCT
	Deceleration : LREAL;
	Jerk	: LREAL;
END_STRUCT
END_TYPE

// Data types/[Internal]/TcNC/_ST_TcNC_StopInfoResponse
{attribute 'conditionalshow'}
TYPE _ST_TcNC_StopInfoResponse :
STRUCT
	StopDistance : LREAL;
	StopTime : LREAL;
END_STRUCT
END_TYPE

// Data types/[Internal]/TcNC/_ST_TcNc_TouchProbeActivation
{attribute 'conditionalshow'}
TYPE _ST_TcNc_TouchProbeActivation :
STRUCT
	TouchProbe 	: UDINT; 	(* number of probe unit 1..4 *)
	Edge		: UDINT; 	(* rising(0) or falling(1) signal edge *)
	Mode		: UDINT;	(* touch probe mode 0=single, 1=continuous *)
	SignalSource	: UDINT;	(* optional physical signal source used by the probe unit *)
	_reserved 	: ARRAY[1..2] OF UDINT;
END_STRUCT
END_TYPE

// Data types/[Internal]/TcNC/_ST_TcNc_TouchProbeDeactivation
{attribute 'conditionalshow'}
TYPE _ST_TcNc_TouchProbeDeactivation :
STRUCT
	TouchProbe 	: UDINT; 	(* number of probe unit 1..4 *)
	Edge		: UDINT; 	(* rising(0) or falling(1) signal edge *)
	_reserved 	: ARRAY[1..4] OF UDINT;
END_STRUCT
END_TYPE

// Data types/[Internal]/TcNC/_ST_TcNc_TouchProbeStatusRequest
{attribute 'conditionalshow'}
TYPE _ST_TcNc_TouchProbeStatusRequest :
STRUCT
	TouchProbe 	: UDINT; 	(* number of probe unit 1..4 *)
	_reserved 	: ARRAY[1..5] OF UDINT;
END_STRUCT
END_TYPE

// Data types/[Internal]/TcNC/_ST_TcNc_TouchProbeStatusResponse
{attribute 'conditionalshow'}
TYPE _ST_TcNc_TouchProbeStatusResponse :
STRUCT
	(* latch status data for the rising signal edge *)
	RisingEdgeActive 		: UDINT;
	RisingEdgeValid		: UDINT;
	RisingEdgeValue 		: LREAL;
	RisingEdgeCounter 	: UDINT;
	_reserved1 			: UDINT;

	(* latch status data for the falling signal edge *)
	FallingEdgeActive 	: UDINT;
	FallingEdgeValid		: UDINT;
	FallingEdgeValue 		: LREAL;
	FallingEdgeCounter	 : UDINT;
	_reserved2 			: UDINT;

	_reserved3 : ARRAY[1..4] OF UDINT;
END_STRUCT
END_TYPE

// Data types/[Internal]/TcNC/_ST_TcNC_UniversalAxisTorqueStartRequest
{attribute 'conditionalshow'}
TYPE _ST_TcNC_UniversalAxisTorqueStartRequest :
STRUCT
	nStartType			: UDINT;			(* axis start TYPE (TORQUECONTINUOUS) *)
	nControlMask		: UDINT;			(* optional: control mask *)

	nMode				: UDINT;			(* optional: mode (ENUM) *)
	nBufferMode			: UDINT;			(* 'buffer mode' OR 'activation mode' FOR 'buffered commands' (first Only ABORTING) *)

	fTorque				: LREAL;			(* target torque [signed]*)
	fTorqueRamp			: LREAL;			(* nc torque ramp *)

	fVelocityLimitHigh	: LREAL;			(* velocity limit high [signed]*)
	fVelocityLimitLow	: LREAL;			(* velocity limit low [signed]*)

	fAcceleration		: LREAL;			(* acceleration (>= 0) *)
	fDeceleration		: LREAL;			(* deceleration (>= 0) *)

	fManualTorque		: LREAL;			(* optional: manual torque (sync value) *)
END_STRUCT
END_TYPE

// Data types/[Internal]/TcNC/_ST_TcNC_UnversalAxisStartRequest
{attribute 'conditionalshow'}
TYPE _ST_TcNC_UnversalAxisStartRequest :
STRUCT
	nStartType	: UDINT;			(* axis start TYPE (ABSOLUT, RELATIV, ENDLESS_PLUS, ENDLESS_MINUS, MODULO_SHORT, MODULO_PLUS, MODULO_MINUS) *)
	nControlMask	: UDINT;			(* optional: control mask *)

	fPosTarget	: LREAL;			(* target position *)
	fVeloRequ	: LREAL;			(* required velocity *)

	fAcc			: LREAL;			(* acceleration (>= 0) *)
	fDec		: LREAL;			(* deceleration (>= 0) *)
	fJerk		: LREAL;			(* jerk (>= 0) *)

	nBufferMode	: UDINT;			(* optional: 'buffer mode' OR 'activation mode' FOR 'buffered commands' (issue #2786) *)
	nReserved	: UDINT;			(* reserved *)
	fBlendingPosition: LREAL;			(* optional: activation position *)

	fVeloStart	: LREAL;			(* optional: start velocity	(0 <= fVeloStart <= fVeloRequ)	Frage: erstmal weglassen ??? *)
	fVeloEnd		: LREAL;			(* optional: end velocity		(0 <= fVeloEnd <= fVeloRequ)	Frage: erstmal weglassen ??? *)
END_STRUCT
END_TYPE

// Data types/[Internal]/TcNC/_ST_TcNC_UnversalAxisStartResponse
{attribute 'conditionalshow'}
TYPE _ST_TcNC_UnversalAxisStartResponse :
STRUCT
	nCmdNo 	: WORD;			(* Continuous actual command number *)
	nCmdState	: WORD;			(* Command state *)
END_STRUCT
END_TYPE

// Data types/[Internal]/_E_ParameterType
{attribute 'conditionalshow'}
TYPE _E_ParameterType :
 (
	PARAMETERTYPE_NOTYPE := 0,
	PARAMETERTYPE_BOOL,
	PARAMETERTYPE_DWORD,
	PARAMETERTYPE_LREAL,
	PARAMETERTYPE_LARGE	// any parameter with size > LREAL; used for LINT or ULINT as well
 );
END_TYPE

// Data types/[Internal]/_E_PhasingState
{attribute 'conditionalshow'}
(* Phasing internal probe states *)
TYPE _E_PhasingState :
 (
	PhasingInactive,
	PhasingActivated,
	PhasingAborted
 );
END_TYPE

// Data types/[Internal]/_E_ReadWriteParameterMode
{attribute 'conditionalshow'}
TYPE _E_ReadWriteParameterMode :
 (
	READWRITEPARAMETERMODE_READ 	:=10,
	READWRITEPARAMETERMODE_WRITE	:= 11
 );
END_TYPE

// Data types/[Internal]/_E_SinusMotionMode
{attribute 'conditionalshow'}
TYPE _E_SinusMotionMode :
(
	eSinusMode_Oscillation := 0,
	eSinusMode_Sequence := 1	
);
END_TYPE

// Data types/[Internal]/_E_TcMC_STATES
{attribute 'conditionalshow'}
TYPE _E_TcMC_STATES :
 (
	STATE_INITIALIZATION  := 100,
	STATE_ORDER,
	STATE_RUNNING,
	STATE_WAITING,
	STATE_MOTIONCOMMANDSLOCKED
 );
END_TYPE

// Data types/[Internal]/_E_TouchProbeState
{attribute 'conditionalshow'}
(* MC_TouchProbe internal probe states *)
TYPE _E_TouchProbeState :
 (
	TouchProbeInactive,
	TouchProbeActivated,
	TouchProbeAborted
 );
END_TYPE

// Data types/[Internal]/_InternalAxisRefData
{attribute 'conditionalshow'}
TYPE _InternalAxisRefData :
STRUCT
	NcCycleCounterAvailable					: BOOL;	(* TRUE if the NcCycleCounter is definitely available on the target system - FALSE if undefined *)

	NcCycleCounter_AtReadStatusCall			: UDINT;	(* current NC cycle counter when calling ReadStatus *)
	LastTaskIndex_AtReadStatusCall 			: BYTE;	(* task index of last recent status update *)
	CounterSameTaskIndex_AtReadStatusCall 	: UINT;	(* counter increments to max 100 if the task index for the status update never changes *)

	PhasingState							: _E_PhasingState;	// KSt 20190703 global handshake for phasing blocks
END_STRUCT
END_TYPE

// Data types/[Internal]/_ST_FunctionBlockResults
{attribute 'conditionalshow'}
TYPE _ST_FunctionBlockResults :
STRUCT
	Done				:	BOOL;
	CommandAborted		:	BOOL;
	Error				:	BOOL;
{attribute 'displaymode':='hex'}
	ErrorID				:	UDINT;
{attribute 'displaymode':='dec'}
	BusyCounter			: 	UDINT; (* busy cycles since triggering the block - 2018-01-24 KSt *)
END_STRUCT
END_TYPE

// Data types/[Internal]/_ST_NcIoOutputData
{attribute 'conditionalshow'}
TYPE _ST_NcIoOutputData :
STRUCT
	ByteOffset				: UDINT;
	BitSelectMask			: UDINT;
	BitValues				: UDINT;
END_STRUCT
END_TYPE

// Data types/[Internal]/_ST_ParaStruct
{attribute 'conditionalshow'}
TYPE _ST_ParaStruct :
STRUCT
	Port		: 	UINT;	(* 2014-07-14 KSt *)
	IndexGroup 	:	UDINT;
	IndexOffset :	UDINT;
	ParaType	:	_E_ParameterType;
	LrealSize	:	UDINT; (* sizeof Lreal data array *)
	LrealOffset	: 	UDINT; (* offset in lreal data array *)
END_STRUCT
END_TYPE

// Data types/Axis Reference/ST_AdsAddress
TYPE ST_AdsAddress :
STRUCT
	NetId	 	: STRING(23);
	Port 		: UINT;
	Channel 	: UINT;
END_STRUCT
END_TYPE

// Data types/BacklashCompensation/ST_BacklashCompensationOptions
TYPE ST_BacklashCompensationOptions :
STRUCT
{attribute 'conditionalshow'}
	_reserved : BOOL;
END_STRUCT
END_TYPE

// Data types/DriveOperationMode/E_DriveOperationMode
TYPE E_DriveOperationMode :
(
	DriveOperationMode_Default						:= 0,   // 0x0000: default => reactivate the nc default op mode (if default mode is known!?!)
	// general operation modes (e.g. CANopen/CoE)
	DriveOperationMode_Torque   					:= 1,  	// 0x0001: torque control 
	DriveOperationMode_Velo1   						:= 2,	// 0x0002: velocity control with feedback 1
	DriveOperationMode_Velo2    					:= 3,   // 0x0003: velocity control with feedback 2
	DriveOperationMode_Pos1  		 	  			:= 4,   // 0x0004: pos control with feedback 1, lag less
	DriveOperationMode_Pos2     					:= 5,   // 0x0005: pos control with feedback 2, lag less
	DriveOperationMode_TorqueAndCommutationAngle	:= 6,   // 0x0006: torque control with commutation angle
	
	// new operation modes using dynamic container (also called 'dynamic MDT' or 'dynamic sync manager')
{attribute 'hide'}
	DriveOperationMode_TorqueDynContainer			:= 17,	// 0x0011: torque ctrl using dynamic container (READ ONLY !!!)
{attribute 'hide'}
	DriveOperationMode_Velo1DynContainer			:= 18,  // 0x0012: velo with ctrl feedback 1 using dynamic container (READ ONLY !!!)
{attribute 'hide'}
	DriveOperationMode_Velo2DynContainer			:= 19,  // 0x0013: velo with ctrl feedback 2 using dynamic container (READ ONLY !!!)
{attribute 'hide'}
	DriveOperationMode_Pos1DynContainer				:= 20,  // 0x0014: pos ctrl with feedback 1 (lag less) using dynamic container (READ ONLY !!!)
{attribute 'hide'}
	DriveOperationMode_Pos2DynContainer				:= 21,  // 0x0015: pos ctrl with feedback 2 (lag less) using dynamic container (READ ONLY !!!)

{attribute 'hide'}
	DriveOperationMode_PositionProfile   			:= 33,   // 0x0021: DS402/CoE specific drive controled Profile position mode
	DriveOperationMode_VelocityMode   				:= 34,   // 0x0022: DS402/CoE specific drive controled velocity mode (VL) (READ ONLY !!!)
{attribute 'hide'}
	DriveOperationMode_VelocityProfile  			:= 35,   // 0x0023: DS402/CoE specific drive controled Profile velocity Mode
{attribute 'hide'}
	DriveOperationMode_TorqueProfile  		 	  	:= 36,   // 0x0024: DS402/CoE specific drive controled Profile torque mode 

	DriveOperationMode_DriveBasedHoming    			:= 38,   // 0x0026: DS402/CoE specific drive controled homing mode
{attribute 'hide'}
	DriveOperationMode_PositionInterpolated    		:= 39,   // 0x0027: DS402/CoE specific drive controled interpolated position mode

	// attention, only for SERCOS/SoE: 
	// 8 special indirect index based operation modes (only for SERCOS/SoE)
	DriveOperationMode_Index0               		:= 100, // 100: SERCOS/SoE operation mode index 0 (primary operation mode 0, s. S-0-0032) 
	DriveOperationMode_Index1               		:= 101, // 101: SERCOS/SoE operation mode index 1 (secondary operation mode 1, s. S-0-0033)
	DriveOperationMode_Index2               		:= 102, // 102: SERCOS/SoE operation mode index 2 (secondary operation mode 2, s. S-0-0034)
	DriveOperationMode_Index3               		:= 103, // 103: SERCOS/SoE operation mode index 3 (secondary operation mode 3, s. S-0-0035)
{attribute 'hide'}
	DriveOperationMode_Index4               		:= 104, // 104: SERCOS/SoE operation mode index 4 (secondary operation mode 4, s. S-0-0284)
{attribute 'hide'}
	DriveOperationMode_Index5               		:= 105, // 105: SERCOS/SoE operation mode index 5 (secondary operation mode 5, s. S-0-0285)
{attribute 'hide'}
	DriveOperationMode_Index6               		:= 106, // 106: SERCOS/SoE operation mode index 6 (secondary operation mode 6, s. S-0-0286)
{attribute 'hide'}
	DriveOperationMode_Index7               		:= 107  // 107: SERCOS/SoE operation mode index 7 (secondary operation mode 7, s. S-0-0287)
) DINT;
END_TYPE

// Data types/DriveOperationMode/ST_DriveOperationModeOptions
TYPE ST_DriveOperationModeOptions :
STRUCT
END_STRUCT
END_TYPE

// Data types/Gearing/E_GearInMultiMasterSyncMode
{attribute 'qualified_only'}
{attribute 'strict'}
TYPE E_GearInMultiMasterSyncMode :
(
	//enum_member := 0
	VELOSYNC, // 0L // 0x0000 0000 (bin: 00000000): velocity synchronization only (0) (DEFAULT)
	POSSYNC1, // 1L // 0x0000 0000 (bin: 00000001): position synchronization (1): catch up position gap after slave dynamic limitation ONLY during synchronous phase 
              // (don’t catch up gap in synchronization phase and when changing gear ratio) => velocity overshoot after dynamic limitation possible
	POSSYNC2  // 2L // 0x0000 0000 (bin: 00000010): position synchronization (2): catch up position gap after slave dynamic limitation during synchronous phase, 
              // synchronization phase and when changing gear ratio => velocity overshoot during synchronization phase possible
);
END_TYPE

// Data types/Gearing/ST_GearInDynOptions
TYPE ST_GearInDynOptions :
STRUCT
	CCVmode : BOOL; (* constant circumference velocity mode *)
END_STRUCT
END_TYPE

// Data types/Gearing/ST_GearInMultiMasterOptions
TYPE ST_GearInMultiMasterOptions :
STRUCT
	AdvancedSlaveDynamics 		: BOOL;
	SyncMode : E_GearInMultiMasterSyncMode;
 //{attribute 'conditionalshow'}
 //	VelocitySynchronizationOnly 	: BOOL;
END_STRUCT
END_TYPE

// Data types/Gearing/ST_GearInOptions
TYPE ST_GearInOptions :
STRUCT
{attribute 'conditionalshow'}	// hidden since 3-2023 KSt because SlaveType is an undocumented option
	SlaveType : _E_TcNC_SlaveTypes;
END_STRUCT
END_TYPE

// Data types/Gearing/ST_GearOutOptions
TYPE ST_GearOutOptions :
STRUCT
{attribute 'conditionalshow'}
	reserved : BOOL;
END_STRUCT
END_TYPE

// Data types/Homing/E_EncoderReferenceMode
TYPE E_EncoderReferenceMode :
(
	ENCODERREFERENCEMODE_DEFAULT 			:= 0,
	ENCODERREFERENCEMODE_PLCCAM 			:= 1,
	ENCODERREFERENCEMODE_HARDWARESYNC 		:= 2,
	ENCODERREFERENCEMODE_HARDWARELATCHPOS 	:= 3,
	ENCODERREFERENCEMODE_HARDWARELATCHNEG 	:= 4,
	ENCODERREFERENCEMODE_SOFTWARESYNC 		:= 5,
	ENCODERREFERENCEMODE_SOFTDRIVELATCHPOS 	:= 6,
	ENCODERREFERENCEMODE_SOFTDRIVELATCHNEG 	:= 7,
{attribute 'conditionalshow'}
	ENCODERREFERENCEMODE_APPLICATION 		:= 20
) UDINT;
END_TYPE

// Data types/Homing/MC_HomingMode
TYPE MC_HomingMode :
 (
	MC_DefaultHoming,	(* default homing as defined in the SystemManager encoder parameters *)
{attribute 'conditionalshow'}
	MC_AbsSwitch,		(* not implemented - Absolute Switch homing plus Limit switches *)
{attribute 'conditionalshow'}
	MC_LimitSwitch,		(* not implemented - Homing against Limit switches *)
{attribute 'conditionalshow'}
	MC_RefPulse,		(* not implemented - Homing using encoder Reference Pulse "Zero Mark" *)
	MC_Direct,			(* Static Homing forcing position from user reference *)
{attribute 'conditionalshow'}
	MC_Absolute,			(* not implemented - Static Homing forcing position from absolute encoder *)
{attribute 'conditionalshow'}
	MC_Block,			(* not implemented - Homing against hardware parts blocking movement *)
	MC_ForceCalibration,	(* set the calibration flag without performing any motion or changing the position *)
	MC_ResetCalibration	(* resets the calibration flag without performing any motion or changing the position *)
 );
END_TYPE

// Data types/Homing/ST_HomingOptions
TYPE ST_HomingOptions :
STRUCT
	ClearPositionLag 		: BOOL;	(* set actual and set position to same value and clear the position lag *)
	
	SearchDirection			: MC_Direction := MC_Direction.MC_Undefined_Direction;
	SearchVelocity			: LREAL;
	SyncDirection			: MC_Direction := MC_Direction.MC_Undefined_Direction;
	SyncVelocity			: LREAL;
	ReferenceMode			: E_EncoderReferenceMode := E_EncoderReferenceMode.ENCODERREFERENCEMODE_DEFAULT;
END_STRUCT
END_TYPE

// Data types/Motion/E_JogMode
TYPE E_JogMode :
 (
	MC_JOGMODE_STANDARD_SLOW,	(* motion with standard jog parameters for slow motion *)
	MC_JOGMODE_STANDARD_FAST,		(* motion with standard jog parameters for fast motion *)
	MC_JOGMODE_CONTINOUS,		 	(* axis moves as long as the jog button is pressed using parameterized dynamics *)
	MC_JOGMODE_INCHING,				(* axis moves for a certain relative distance *)
	MC_JOGMODE_INCHING_MODULO		(* axis moves for a certain relative distance - stop position is rounded to the distance value *)
 );
END_TYPE

// Data types/Motion/E_PositionType
TYPE E_PositionType :
(
	POSITIONTYPE_ABSOLUTE	:= 1,	(*Absolute position*)
	POSITIONTYPE_RELATIVE,		(*Relative position*)
	POSITIONTYPE_MODULO		:= 5	(*Modulo position*)
) UINT;
END_TYPE

// Data types/Motion/MC_BufferMode
TYPE MC_BufferMode :
 (
	MC_Aborting			:= 16#00,
	MC_Buffered			:= 16#01,
	MC_BlendingLow		:= 16#12,
	MC_BlendingPrevious	:= 16#13,
	MC_BlendingNext		:= 16#14,
	MC_BlendingHigh		:= 16#15
 ) UINT;
END_TYPE

// Data types/Motion/MC_Direction
TYPE MC_Direction :
(
	MC_Positive_Direction := 1,
	MC_Shortest_Way ,
	MC_Negative_Direction,
	MC_Current_Direction,
	MC_Undefined_Direction := 128
);
END_TYPE

// Data types/Motion/ST_MoveOptions
TYPE ST_MoveOptions :
STRUCT
	(* Command activation at defined ActivationPosition - extends the buffer mode when enabled *)
	EnableBlendingPosition : BOOL;
	BlendingPosition : LREAL;

	(* velocity profile options - instantaneous speed change at the beginning and at the end of the profile *)
	StartVelocity : LREAL;
	EndVelocity : LREAL;	
	
	(* PositionAreaMonitoring, TargetPositionMonitoring and StopMonitoring can be ignored using this flag - 20190311 *)
	IgnorePositionMonitoring : BOOL; 
	
	(* PositionAreaMonitoring, TargetPositionMonitoring can be enabled for MC_Stop and MC_Halt commands - 20191010 *)
	(* Monitoring can just be enabled if the monitoring parameters of the axis are enabled as well *)
	(* The default is no monitoring for both commands even if monitoring options are enabled by axis parameters *)
	EnableStopPositionMonitoring : BOOL;
END_STRUCT
END_TYPE

// Data types/Nc Process Data/E_NcIoDevice
TYPE E_NcIoDevice :
(
	NcIoDeviceDrive := 0,
	NcIoDeviceEncoder := 1
);
END_TYPE

// Data types/Nc Process Data/E_NcIoOutput
TYPE E_NcIoOutput :
(
	NcIoOutputnCtrl1 := 0,
	NcIoOutputnCtrl2 := 1,
	NcIoOutputnCtrl3 := 2,
	NcIoOutputnCtrl4 := 3,
	NcIoOutputnCtrl5 := 4,
	NcIoOutputnCtrl6 := 5,
	NcIoOutputnCtrl7 := 6,
	NcIoOutputnCtrl8 := 7,
	NcIoOutputnDataOut1 := 8,
	NcIoOutputnDataOut2 := 9,
	NcIoOutputnDataOut3 := 10,
	NcIoOutputnDataOut4 := 11,
	NcIoOutputnDataOut5 := 12,
	NcIoOutputnDataOut6 := 13
);
END_TYPE

// Data types/Phasing/E_PhasingType
TYPE E_PhasingType :
 (
	NC_PHASINGTYPE_ABSOLUTE 	:= 1,
	NC_PHASINGTYPE_RELATIVE 	:= 2,
	NC_PHASINGTYPE_STOP 		:= 4096
 ) UINT;
END_TYPE

// Data types/Phasing/ST_PhasingOptions
TYPE ST_PhasingOptions :
STRUCT
{attribute 'conditionalshow'}
	_reserved : BOOL;
END_STRUCT
END_TYPE

// Data types/Position Correction/E_AxisPositionCorrectionMode
TYPE E_AxisPositionCorrectionMode :
 (
	POSITIONCORRECTION_MODE_UNLIMITED,	(* no limitation - pass correction immediately *)
	POSITIONCORRECTION_MODE_FAST,		(* limitatation to maximum position change per cycle *)
	POSITIONCORRECTION_MODE_FULLLENGTH	(* limitation uses full length to adapt to correction in small steps *)
 );
END_TYPE

// Data types/Position Correction/ST_PositionCompensationOptions
TYPE ST_PositionCompensationOptions :
STRUCT
{attribute 'conditionalshow'}
	_reserved : BOOL;
END_STRUCT
END_TYPE

// Data types/Position Correction/ST_PositionCompensationTableElement
TYPE ST_PositionCompensationTableElement :
STRUCT
	Position		: LREAL;	(* uncorrected position value (e.g. SetPos) *)
	Compensation	: LREAL;	(* additive compensation value *)
END_STRUCT
END_TYPE

// Data types/Position Correction/ST_PositionCompensationTableParameter
TYPE ST_PositionCompensationTableParameter :
STRUCT
	MinPosition			: LREAL;		(* compensation starts with this position *)
	MaxPosition			: LREAL;		(* compensation ends with this position *)
	NoOfTableElements	: UDINT;		(* number of entries in table *)
	Direction			: E_WorkDirection := WorkDirectionBoth;	(* compensation is just working in the selected working direction *)
	Modulo				: BOOL ;		(* FALSE: linear axis, TRUE: modulo axis with cyclic period (e.g. 360 degree) *)
(*	TableType			: E_CompensationTableType:=TableType1DEquidistant; *)	(* NOT NEEDED YET *)
END_STRUCT
END_TYPE

// Data types/SelectControlLoop/E_SelectControlLoopType
TYPE E_SelectControlLoopType :
(
	SelectControlLoopType_Undefined,			(* NICHT DEFINIERT *)
	SelectControlLoopType_Standard,				(* Einfaches Umschalten (ähnlich einem Achsreset) (STANDARD) *)
	SelectControlLoopType_InternalSyncValue,	(* Umschalten/Aufsynchronisieren mittels I/D-Anteil des Reglers auf einen internen Initialwert (ruckfrei/stoßfrei) *)
	SelectControlLoopType_UserSyncValue			(* Umschalten/Aufsynchronisieren mittels I/D-Anteil des Reglers auf einen parametrierbaren Initialwert *)
) UDINT;
END_TYPE

// Data types/SelectControlLoop/ST_SelectControlLoop
{attribute 'conditionalshow'}
TYPE ST_SelectControlLoop :
STRUCT
	EncoderIndex		: UDINT;	(* 0, 1, 2... *)
	SelectType 			: UDINT;
	SyncValue 			: LREAL;
	ExtSetPointGen 		: UDINT;
END_STRUCT
END_TYPE

// Data types/Status and Parameter/E_AxisErrorCodes
(* for details: see TwinCAT Information System*)
TYPE E_AxisErrorCodes : (
		MC_ERROR_NO_ERROR := 0,
(*		MC_ERROR_NO_ORDER,		deleted 15.07.2005 KSt *)
(*		MC_ERROR_OVERRIDE,		deleted 15.07.2005 KSt *)
(*		MC_ERROR_LOW_VELOCITY,	deleted 15.07.2005 KSt *)
		MC_ERROR_AXIS_HAS_BEEN_STOPPED		:= 16#4B00,
		MC_ERROR_AXIS_CAN_NOT_BE_STARTED	:= 16#4B01,
		MC_ERROR_CONTROLMODE_NOT_ALLOWED	:= 16#4B02,
		MC_ERROR_AXIS_IS_NOT_MOVING			:= 16#4B03,
		MC_ERROR_WRONG_MODE					:= 16#4B04,
		MC_ERROR_COMMAND_NOT_ALLOWED		:= 16#4B05,
		MC_ERROR_PARAMETER_NOT_CORRECT		:= 16#4B06,
		MC_ERROR_TARGETPOS_TIMEOUT			:= 16#4B07,
		MC_ERROR_AXIS_IN_PROTECTED_MODE		:= 16#4B08,
		MC_ERROR_AXIS_IS_NOT_READY				:= 16#4B09,
		MC_ERROR_CALIBRATION_ERROR			:= 16#4B0A,
		MC_ERROR_INVALID_TOUCH_PROBE			:= 16#4B0B,
		MC_ERROR_TOUCH_PROBE_DEACTIVATED	:= 16#4B0C,
		MC_ERROR_STATE_FEEDBACK_TIMEOUT		:= 16#4B0D,
		MC_ERROR_SUPPLEMENT_NOT_INSTALLED	:= 16#4B0E,
		MC_ERROR_NCCYCLECOUNTERUPDATE		:= 16#4B0F,
		(*======================================================================	*)
		(*	4B0F 	timeout terminal register access									*)
		(*======================================================================	*)
		(* 	4B10 .. 4B2F used in NCI context 											*)
		(*======================================================================	*)
		(* 	4B30 .. 4B3F used in TcMcCam - MC_NC_TableErrorCodes					*)
		(*======================================================================	*)
		(* 	4B40 .. 4B4F used in TcNc.lib for programming KL25xx terminals 				*)	(*
		ERRORCODE_INVALIDPARAMETER	 				:= 16#4B06;
		ERRORCODE_TIMEOUTREGISTERCOMMUNICATION 	:= 16#4B0F;	// ATTENTION see MC_ERROR_NCCYCLECOUNTERUPDATE //
		ERRORCODE_TERMINALTYPENOTSUPPORTED 		:= 16#4B40;
		ERRORCODE_WRITEERROR							:= 16#4B41;
		ERRORCODE_AXISENABLED							:= 16#4B42;
		ERRORCODE_PARAMSIZE							:= 16#4B43;
		ERRORCODE_PARAMPOS							:= 16#4B44;
		ERRORCODE_TCNCNOTIMPL							:= 16#4B45;
		*)
		(*======================================================================	*)
		(* 	4B50 .. 4B59 used in TcRemoteSync.lib									*)
		(*======================================================================	*)
		(* 	4B5A .. 4B5F 		FREE												*)
		(*======================================================================	*)
		(* 	4B60 .. 4B6F used in TcMC for buffered commands  *)
		MC_ERROR_BUFFERED_COMMAND_NOT_STARTED			:= 16#4B60,
		MC_ERROR_BUFFERED_COMMAND_MONITORING_IMPOSSIBLE	:= 16#4B61,
		MC_ERROR_BUFFERED_COMMAND_ERRORID_NOT_AVAILABLE	:= 16#4B62,
		MC_ERROR_BUFFERED_COMMAND_NO_STATE_FEEDBACK		:= 16#4B63,
		MC_ERROR_BUFFERMODE_NOT_SUPPORTED					:= 16#4B64,
		MC_ERROR_BUFFERED_COMMAND_CMDNOZERO				:= 16#4B65,
		MC_ERROR_BUFFCMD_MONITRNGIMPOSS_FBNOTCALLEDCYC	:= 16#4B66,	(* command monitoring impossible because function block was not cyclically called - alternative error to 4B61 *)
		MC_ERROR_FUNCTIONBLOCK_NOT_CYCLICALLY_CALLED 		:= 16#4B6F,	(* function block was not cyclically called *)

		(*======================================================================	*)
		(* 	4B70 .. 4B70 used in TcMC for I/O related errors *)
		MC_ERROR_TERMINALFEEDBACK								:= 16#4B70,	(* UNUSED ??? *)
		(*======================================================================	*)
		(* 	4B71 .. 4B8F used in TcPlcInterpolation.Lib  *)
		(*======================================================================	*)
		(* 	4B90 .. 4B9F used in Tc2_MC2_AdvancedHoming.Lib (TC3 only) *)
		(*======================================================================	*)


(*		MC_ERROR_FUNCTION_IS_BUSY := 16#4B99	*)

		MC_ERROR_INVALIDREFERENCE := 16#8189 	(* 2020-09-17 KSt used for checks of reference variables *)
		) UINT;
END_TYPE

// Data types/Status and Parameter/E_DisableMode
TYPE E_DisableMode :
(
	DisableModeHold		:= 0,		(* hold on the last output value (default) *)
	DisableModeReset	:= 1		(* reset the output value to zero (jump to zero) *)
(*	DisbaleModeRamp		:= 2 *)		(* ramp down the output to zero (NOT NEEDED YET) *)
);
END_TYPE

// Data types/Status and Parameter/E_NcAxisType
TYPE E_NcAxisType :
(
	NcAxisType_undefined						:= 0,	
	NcAxisType_Continious						:= 1,   // Kontinuierliche Achse (auch SERCOS)
	NcAxisType_Discrete_TwoSpeed				:= 2,   // Diskrete Achse (Eil/Schleich-Achse)
	NcAxisType_LowCostStepper_DigIO				:= 3,   // Schrittmotor Achse (ohne PWM Klemme KL2502/30 und ohne Pulse-Train KL2521)
	NcAxisType_Encoder							:= 5,   // Encoder Achse
	NcAxisType_Hydraulic						:= 6,   // Kontinuierliche Achse mit Betriebsartumschaltung fur Positions-/Druck-Regelung
	NcAxisType_TimeGenerator					:= 7,   // Time Base Generator 
	NcAxisType_Specific							:= 100
) DWORD;
END_TYPE

// Data types/Status and Parameter/E_NcDriveType
TYPE E_NcDriveType :
(
	NcDriveType_undefined						:= 0,
	NcDriveType_M2400_DAC1						:= 1,
	NcDriveType_M2400_DAC2						:= 2,
	NcDriveType_M2400_DAC3						:= 3,
	NcDriveType_M2400_DAC4						:= 4,
	NcDriveType_KL4XXX							:= 5,	// MDP 252/253: KL4xxx, PWM KL2502_30K (Frq-Cnt-Impuls-Modus), KL4132 (16 Bit), Pulse-Train KL2521, IP2512
	NcDriveType_KL4XXX_NonLinear				:= 6,	// MDP 252/253: Analog-Typ für nichtlineare Kennlinie
	NcDriveType_Discete_TwoSpeed				:= 7,
	NcDriveType_Stepper							:= 8,
	NcDriveType_Sercos							:= 9,
	NcDriveType_KL5051							:= 10,	// MDP 510: BISSI Drive KL5051 mit 32 Bit (siehe KL4XXX)
	NcDriveType_AX2000_B200						:= 11,	// AX2000-B200 Lightbus, Inkremental mit 32 Bit (AX2000)
	NcDriveType_ProfiDrive						:= 12,  // Inkremental mit 32 Bit 
	NcDriveType_Universal						:= 13,  // Variable Bitmaske (max. 32 Bit, signed value)
	NcDriveType_NcBackplane						:= 14,  // Variable Bitmaske (max. 32 Bit, signed value)
	NcDriveType_CANopen_Lenze					:= 15,  // CANopen Lenze (max. 32 Bit, signed value)
	NcDriveType_CANopen_DS402_MDP742			:= 16,  // MDP 742 (DS402): CANopen und EtherCAT (AX2000-B510, AX2000-B1x0, EL7201, AX8000)
	NcDriveType_AX2000_B900						:= 17,  // AX2000-B900 Ethernet (max. 32 Bit, signed value)
//	NcDriveType_AX2000_B310						:= 18,  // AX2000-B310 Profibus (nie implementiert worden!!!)
	NcDriveType_KL2531_Stepper					:= 20,  // Schrittmotorklemme KL2531/KL2541
	NcDriveType_KL2532_DC						:= 21,  // 2-Kanal-DC-Motor-Endstufe (2-channel DC motor stage) KL2532/KL2542, 2-Kanal-PWM-DC-Motorendstufe KL2535/KL2545
	NcDriveType_TCOM							:= 22,  // TCOM Drive -> Interface to Soft Drive
	NcDriveType_MDP_733							:= 23,  // MDP 733: Modular Device Profile MDP 733 for DC (e.g. EL7332/EL7342) (20.02.09)
	NcDriveType_MDP_703							:= 24   // MDP 703: Modular Device Profile MDP 703 for stepper (e.g. EL7031/EL7041) 
) DWORD;
END_TYPE

// Data types/Status and Parameter/E_NcEncoderType
TYPE E_NcEncoderType :
(
	NcEncoderType_undefined							:= 0,
	NcEncoderType_Simulation						:= 1,	// Simulation
	NcEncoderType_ABS_M3000							:= 2,   // Absolut mit 24 und 25 Bit sowie 12 und 13 Bit Single Turn Encoder (M3000)
	NcEncoderType_INC_M31X0							:= 3,   // Inkremental mit 24 Bit (M31x0, M3200, M3100, M2000)
	NcEncoderType_INC_KL5101						:= 4,   // MDP 511: Inkremental mit 16 Bit und Latch (MDP511: EL7041, EL5101, EL5151, EL2521, EL5021(SinCos); KL5101, IP5109, KL5111)
	NcEncoderType_ABS_KL5001_SSI					:= 5,   // MDP 500/501: Absolut SSI mit 24 Bit (KL5001, IP5009)(MDP 501: EL5001)
	NcEncoderType_INC_KL5051						:= 6,   // MDP 510: Absolut/Inkremental BISSI mit 16 Bit (KL5051, PWM KL2502_30K (Frq-Cnt-Impuls-Modus), Pulse-Train KL2521, IP2512 ) 
	NcEncoderType_ABS_KL30XX						:= 7,   // Absolut Analog Eingang mit 16 Bit (KL30xx)
	NcEncoderType_INC_Sercos_P						:= 8,   // SERCOS "Encoder" POS
	NcEncoderType_INC_Sercos_PV						:= 9,   // SERCOS "Encoder" POS und VELO
	NcEncoderType_INC_Binary						:= 10,  // Binaerer Inkremental Encoder (0/1)
	NcEncoderType_ABS_M2510							:= 11,  // Absolut Analog Eingang mit 12 Bit (M2510)
	NcEncoderType_ABS_FOX50			    			:= 12,  // T&R Fox 50 Modul (24 Bit Absolut (SSI))
	NcEncoderType_ABS_HYDRAULIC_FORCE				:= 13,  // MMW-Typ: Kraftermittlung aus Pa, Pb, Aa, Ab
	NcEncoderType_INC_AX2000_B200	  				:= 14,  // Inkremental AX2000-B200 Lightbus mit 16/20 Bit (AX2000)
	NcEncoderType_INC_PROFIDRIVE	    			:= 15,  // Inkremental mit 32 Bit
	NcEncoderType_INC_UNIVERSAL		   				:= 16,  // Inkremental mit variabler Bitmaske (max. 32 Bit)
	NcEncoderType_INC_NCBACKPLANE	  				:= 17,  // Inkremental NC Rückwand
	NcEncoderType_INC_CANOPEN_LENZE					:= 18,  // Inkremental CANopen Lenze
	NcEncoderType_INC_CANOPEN_DS402_MDP513_MDP742 	:= 19,  // MDP 513 / MDP 742 (DS402): CANopen und EtherCAT (AX2000-B510, AX2000-B1x0, EL7201, EL5032/32Bit)
	NcEncoderType_INC_AX2000_B900	  				:= 20,  // Inkremental AX2000-B900 Ethernet
	NcEncoderType_INC_KL5151		    			:= 21,  // Inkremental mit 32 Bit Zaehler und int.+ ext. 32 Bit Latch (KL5151_0000) (nur umschaltbar), die 2-kanalige KL5151_0050 hat kein Latch !
//	NcEncoderType_INC_AX2000_B310	  				:= 22,  // Inkremental AX2000-B310 Profibus (nie implementiert worden!!!)
	NcEncoderType_INC_IP5209						:= 24,	// Inkremental mit 32 Bit Zaehler und int. 32 Bit Latch (IP5209)
	NcEncoderType_INC_KL2531_Stepper				:= 25,  // Inkremental mit 16 Bit Zaehler und int.+ext. 16 Bit Latch (nur umschaltbar) (Schrittmotorklemme KL2531/KL2541)
	NcEncoderType_INC_KL2532_DC						:= 26,  // Inkremental mit 16 Bit Zaehler und ext. 16 Bit Latch (nur umschaltbar) (2-Kanal-DC-Motor-Endstufe KL2532/KL2542), 2-Kanal-PWM-DC-Motorendstufe KL2535/KL2545
	NcEncoderType_INC_TIMEBASEGENERATOR				:= 27,  // Time Base Generator
	NcEncoderType_INC_TCOM							:= 28,  // TCOM Encoder -> Interface to Soft Drive Encoder
	NcEncoderType_INC_CANOPEN_MDP513_64BIT			:= 29,  // MDP 513 (DS402, EnDat2.2, 64 Bit): EL5032/64Bit
	NcEncoderType_SPECIFIC							:= 100
) DWORD;
END_TYPE

// Data types/Status and Parameter/E_ReadMode
TYPE E_ReadMode :
 (
 	READMODE_ONCE	:= 1,
	READMODE_CYCLIC
 );
END_TYPE

// Data types/Status and Parameter/E_SetScalingFactorMode
TYPE E_SetScalingFactorMode :
 (
	ENCODERSCALINGMODE_ABSOLUTE	:= 1,
	ENCODERSCALINGMODE_RELATIVE	:=2
 ) UINT;
END_TYPE

// Data types/Status and Parameter/E_WorkDirection
TYPE E_WorkDirection :
(
	WorkDirectionNone		:= 0,
	WorkDirectionBoth		:= 1,
	WorkDirectionPositive	:= 2,
	WorkDirectionNegative	:= 3
);
END_TYPE

// Data types/Status and Parameter/MC_AxisParameter
TYPE MC_AxisParameter : (
(*			PLCopen specific parameters *)			(* Index-Group 0x4000 + ID*)
(*  1 *)		CommandedPosition := 1,		(* lreal *)	(* taken from NcToPlc *)
(*  2 *)		SWLimitPos,					(* lreal *)	(* IndexOffset= 16#0001_000E *)
(*  3 *)		SWLimitNeg,					(* lreal *)	(* IndexOffset= 16#0001_000D *)
(*  4 *)		EnableLimitPos,				(* bool *)	(* IndexOffset= 16#0001_000C *)
(*  5 *)		EnableLimitNeg,				(* bool *)	(* IndexOffset= 16#0001_000B *)
(*  6 *)		EnablePosLagMonitoring,		(* bool *)	(* IndexOffset= 16#0002_0010 *)
(*  7 *)		MaxPositionLag,				(* lreal *)	(* IndexOffset= 16#0002_0012 *)
(*  8 *)		MaxVelocitySystem,			(* lreal *)	(* IndexOffset= 16#0000_0027 *)
(*  9 *)		MaxVelocityAppl,				(* lreal *)	(* IndexOffset= 16#0000_0027 *)
(* 10 *)		ActualVelocity,				(* lreal *)	(* taken from NcToPlc *)
(* 11 *)		CommandedVelocity,			(* lreal *)	(* taken from NcToPlc *)
(* 12 *)		MaxAccelerationSystem,		(* lreal *)	(* IndexOffset= 16#0000_0101 *)
(* 13 *)		MaxAccelerationAppl,			(* lreal *)	(* IndexOffset= 16#0000_0101 *)
(* 14 *)		MaxDecelerationSystem,		(* lreal *)	(* IndexOffset= 16#0000_0102 *)
(* 15 *)		MaxDecelerationAppl,			(* lreal *)	(* IndexOffset= 16#0000_0102 *)
(* 16 *)		MaxJerkSystem,				(* lreal *)	(* IndexOffset= 16#0000_0103 *)
(* 17 *)		MaxJerkAppl,					(* lreal *)	(* IndexOffset= 16#0000_0103 *)

(*			Beckhoff specific parameters *)		 	(* Index-Group 0x4000 + ID*)
			AxisId	:=	1000,				(* lreal *)	(* IndexOffset= 16#0000_0001 *)
			AxisVeloManSlow,				(* lreal *)	(* IndexOffset= 16#0000_0008 *)
			AxisVeloManFast,				(* lreal *)	(* IndexOffset= 16#0000_0009 *)
			AxisVeloMax,					(* lreal *)	(* IndexOffset= 16#0000_0027 *)
			AxisAcc,						(* lreal *)	(* IndexOffset= 16#0000_0101 *)
			AxisDec,						(* lreal *)	(* IndexOffset= 16#0000_0102 *)
			AxisJerk,						(* lreal *)	(* IndexOffset= 16#0000_0103 *)
			MaxJerk,						(* lreal *)	(* IndexOffset= 16#0000_0103 *)
			AxisMaxVelocity,				(* lreal *)	(* IndexOffset= 16#0000_0027 *)
			AxisRapidTraverseVelocity,		(* lreal *)	(* IndexOffset= 16#0000_000A *)
			AxisManualVelocityFast,			(* lreal *)	(* IndexOffset= 16#0000_0009 *)
			AxisManualVelocitySlow,			(* lreal *)	(* IndexOffset= 16#0000_0008 *)
			AxisCalibrationVelocityForward,	(* lreal *)	(* IndexOffset= 16#0000_0006 *)
			AxisCalibrationVelocityBackward,(* lreal *)	(* IndexOffset= 16#0000_0007 *)
			AxisJogIncrementForward,		(* lreal *)	(* IndexOffset= 16#0000_0018 *)
			AxisJogIncrementBackward,		(* lreal *)	(* IndexOffset= 16#0000_0019 *)
			AxisEnMinSoftPosLimit,			(* bool *)	(* IndexOffset= 16#0001_000B *)
			AxisMinSoftPosLimit,			(* lreal *)	(* IndexOffset= 16#0001_000D *)
			AxisEnMaxSoftPosLimit,			(* bool *)	(* IndexOffset= 16#0001_000C *)
			AxisMaxSoftPosLimit,			(* lreal *)	(* IndexOffset= 16#0001_000E *)
			AxisEnPositionLagMonitoring,	(* bool *)	(* IndexOffset= 16#0002_0010 *)
			AxisMaxPosLagValue,				(* lreal *)	(* IndexOffset= 16#0002_0012 *)
			AxisMaxPosLagFilterTime,		(* lreal *)	(* IndexOffset= 16#0002_0013 *)
			AxisEnPositionRangeMonitoring,	(* bool *)	(* IndexOffset= 16#0000_000F *)
			AxisPositionRangeWindow,		(* lreal *)	(* IndexOffset= 16#0000_0010 *)
			AxisEnTargetPositionMonitoring,	(* bool *)	(* IndexOffset= 16#0000_0015 *)
			AxisTargetPositionWindow,		(* lreal *)	(* IndexOffset= 16#0000_0016 *)
			AxisTargetPositionMonitoringTime,(* lreal *)(* IndexOffset= 16#0000_0017 *)
			AxisEnInTargetTimeout,			(* bool *)	(* IndexOffset= 16#0000_0029 *)
			AxisInTargetTimeout,			(* lreal *)	(* IndexOffset= 16#0000_002A *)
			AxisEnMotionMonitoring,			(* bool *)	(* IndexOffset= 16#0000_0011 *)
			AxisMotionMonitoringWindow,		(* lreal *)	(* IndexOffset= 16#0000_0028 *)
			AxisMotionMonitoringTime,		(* lreal *)	(* IndexOffset= 16#0000_0012 *)
			AxisDelayTimeVeloPosition,		(* lreal *)	(* IndexOffset= 16#0000_0104 *)
			AxisEnLoopingDistance,			(* bool *)	(* IndexOffset= 16#0000_0013 *)
			AxisLoopingDistance,			(* lreal *)	(* IndexOffset= 16#0000_0014 *)
			{attribute 'hide'}	// old backlash compensation hidden since 9-2020, KST
			AxisEnBacklashCompensation,		(* bool *)	(* IndexOffset= 16#0000_002B *)
//			{attribute 'hide'}	// old backlash compensation hidden since 9-2020, KST
//			backlash compensation visible again since 3-2023, KST
			AxisBacklash,					(* lreal *)	(* IndexOffset= 16#0000_002C *)
			AxisEnDataPersistence,			(* bool *)	(* IndexOffset= 16#0000_0030 *)
			AxisRefVeloOnRefOutput,			(* lreal *)	(* IndexOffset= 16#0003_0101 *)
			AxisOverrideType,				(* lreal *)	(* IndexOffset= 16#0000_0105 *)
			(* new since 4/2007 *)
			AxisEncoderScalingFactor,		(* lreal *)	(* IndexOffset= 16#0001_0006 *)
			AxisEncoderOffset,				(* lreal *)	(* IndexOffset= 16#0001_0007 *)
			AxisEncoderDirectionInverse,	(* bool *)	(* IndexOffset= 16#0001_0008 *)
			AxisEncoderMask,				(* dword *) (* IndexOffset= 16#0001_0015 *)
			AxisEncoderModuloValue,			(* lreal *)	(* IndexOffset= 16#0001_0009 *)
			AxisModuloToleranceWindow,		(* lreal *)	(* IndexOffset= 16#0001_001B *)
			AxisEnablePosCorrection,		(* bool *)	(* IndexOffset= 16#0001_0016 *)
			AxisPosCorrectionFilterTime,	(* lreal *)	(* IndexOffset= 16#0001_0017 *)
			AxisUnitInterpretation,			(* lreal *)	(* IndexOffset= 16#0000_0026 *)	(* added 5/20/2008 KSt *)
			(* new since 1/2010 *)
			AxisMotorDirectionInverse,		(* bool *)	(* IndexOffset= 16#0003_0006 *)
			(* new since 1/2011 *)
			AxisCycleTime,					(* lreal *)	(* IndexOffset= 16#0000_0004 *)
			(* new since 5/2011 *)
			AxisFastStopSignalType,			(* dword *)(* IndexOffset= 16#0000_001E *)
			AxisFastAcc,					(* lreal *)	(* IndexOffset= 16#0000_010A *)
			AxisFastDec,					(* lreal *)	(* IndexOffset= 16#0000_010B *)
			AxisFastJerk,					(* lreal *)	(* IndexOffset= 16#0000_010C *)
			(* new since 1/2012 *)
			AxisEncoderScalingNumerator,	(* lreal *)	(* IndexOffset= 16#0001_0023 - available in Tc3 *)
			AxisEncoderScalingDenominator,	(* lreal *)	(* IndexOffset= 16#0001_0024 - available in Tc3 *)
 			(* new since 7/2016 *)
			AxisMaximumAcceleration,		(* lreal *)	(* IndexOffset= 16#0000_00F1 - available in Tc3 *)
			AxisMaximumDeceleration,		(* lreal *)	(* IndexOffset= 16#0000_00F2 - available in Tc3 *)
			AxisVeloJumpFactor,				(* lreal *)	(* IndexOffset= 16#0000_0106 *)
			AxisToleranceBallAuxAxis,		(* lreal *)	(* IndexOffset= 16#0000_0108 *)
			AxisMaxPositionDeviationAuxAxis,(* lreal *)	(* IndexOffset= 16#0000_0109 *) 
			AxisErrorPropagationMode,		(* dword *) (* IndexOffset= 16#0000_001A *)
			AxisErrorPropagationDelay,		(* lreal *)	(* IndexOffset= 16#0000_001B *) 
			AxisCoupleSlaveToActualValues,	(* bool *)	(* IndexOffset= 16#0000_001C *)
			AxisAllowMotionCmdToSlaveAxis,	(* bool *)	(* IndexOffset= 16#0000_0020 *)
			AxisAllowMotionCmdToExtSetAxis,	(* bool *)	(* IndexOffset= 16#0000_0021 *)
			AxisEncoderSubMask,				(* dword *) (* IndexOffset= 16#0001_0108 *)
			AxisEncoderReferenceSystem,		(* dword *) (* IndexOffset= 16#0001_0019 *)
			AxisEncoderPositionFilterPT1,	(* lreal *)	(* IndexOffset= 16#0001_0010 *)
			AxisEncoderVelocityFilterPT1,	(* lreal *)	(* IndexOffset= 16#0001_0011 *)
			AxisEncoderAccelerationFilterPT1,(* lreal *)(* IndexOffset= 16#0001_0012 *)
			AxisEncoderMode,				(* dword *) (* IndexOffset= 16#0001_000A *)
			AxisEncoderHomingInvDirCamSearch,(* bool *) (* IndexOffset= 16#0001_0101 *)
			AxisEncoderHomingInvDirSyncSearch,(* bool *)(* IndexOffset= 16#0001_0102 *)
			AxisEncoderHomingCalibValue,	(* lreal *) (* IndexOffset= 16#0001_0103 *)
			AxisEncoderReferenceMode,		(* dword *) (* IndexOffset= 16#0001_0107 *)		
			AxisRefVeloOutputRatio,			(* lreal *) (* IndexOffset= 16#0003_0102 *)
			AxisDrivePositionOutputScaling,	(* lreal *) (* IndexOffset= 16#0003_0109 *)
			AxisDriveVelocityOutputScaling,	(* lreal *) (* IndexOffset= 16#0003_0105 *)
			AxisDriveVelocityOutputDelay,	(* lreal *) (* IndexOffset= 16#0003_010D *)
			AxisDriveMinOutputLimitation,	(* lreal *) (* IndexOffset= 16#0003_000B *)
			AxisDriveMaxOutputLimitation,	(* lreal *) (* IndexOffset= 16#0003_000C *)
			AxisTorqueInputScaling,			(* lreal *) (* IndexOffset= 16#0003_0031 - available in Tc3 *)
			AxisTorqueInputFilterPT1,		(* lreal *) (* IndexOffset= 16#0003_0032 - available in Tc3 *)
			AxisTorqueDerivationInputFilterPT1,	(* lreal *) (* IndexOffset= 16#0003_0033 - available in Tc3 *)
			AxisTorqueOutputScaling,		(* lreal *) (* IndexOffset= 16#0003_010B *)
			AxisTorqueOutputDelay,			(* lreal *) (* IndexOffset= 16#0003_010F *)
			AxisAccelerationOutputScaling,	(* lreal *) (* IndexOffset= 16#0003_010A *)
			AxisAccelerationOutputDelay,	(* lreal *) (* IndexOffset= 16#0003_010E *)
			AxisDrivePosOutputSmoothFilterType, (* dword *) (* IndexOffset= 16#0003_0110 *)
			AxisDrivePosOutputSmoothFilterTime,	(* lreal *) (* IndexOffset= 16#0003_0111 *)
			AxisDrivePosOutputSmoothFilterOrder,(* dword *) (* IndexOffset= 16#0003_0112 *)
			AxisDriveMode,					(* dword *) (* IndexOffset= 16#0003_000A *)
			AxisDriftCompensationOffset,	(* lreal *) (* IndexOffset= 16#0003_0104 *)
			AxisPositionControlKv,			(* lreal *) (* IndexOffset= 16#0002_0102 *)
			AxisCtrlVelocityPreCtrlWeight,	(* lreal *) (* IndexOffset= 16#0002_000B *)
			AxisControllerMode,				(* dword *) (* IndexOffset= 16#0002_000A *)
			AxisCtrlAutoOffset,				(* bool  *) (* IndexOffset= 16#0002_0110 *)
			AxisCtrlAutoOffsetTimer,		(* lreal *) (* IndexOffset= 16#0002_0115 *)
			AxisCtrlAutoOffsetLimit,		(* lreal *) (* IndexOffset= 16#0002_0114 *)
			AxisSlaveCouplingControlKcp,	(* lreal *) (* IndexOffset= 16#0002_010F *)
			AxisCtrlOutputLimit,			(* lreal *) (* IndexOffset= 16#0002_0100 *)
			(* new since 6/2018 *)
			AxisFadingAccleration,			(* lreal *) (* IndexOffset= 16#0000_001D *)
			(* new since 6/2022 *)
			AxisUserDataIdxOffs,			(* dword *) (* IndexOffset= 16#0000_010D *)
			
(*			Beckhoff specific axis status information - READ ONLY *)	(* Index-Group 0x4100 + ID*)
			AxisTargetPosition	:= 2000,	(* lreal *)	(* IndexOffset= 16#0000_0013 *)
			AxisRemainingTimeToGo,			(* lreal *)	(* IndexOffset= 16#0000_0014 *)
			AxisRemainingDistanceToGo,		(* lreal *)	(* IndexOffset= 16#0000_0022, 16#0000_0042 *)

(*			Beckhoff specific axis functions *)
			(* read/write gear ratio of a slave - added 6/08/2008 KSt *)
			AxisGearRatio		:= 3000,	(* lreal *) 	(* read:IdxGrp=0x4100+ID, IdxOffs=16#0000_0022, write:IdxGrp=0x4200+ID, IdxOffs=16#0000_0042 *)

(*			Beckhoff specific other parameters *)
			(* new since 1/2011 *)
			NcSafCycleTime 		:= 4000,	(* lreal *)	(* IndexOffset= 16#0000_0010 *)
			NcSvbCycleTime,					(* lreal *)	(* IndexOffset= 16#0000_0012 *)
			
(*			large or structured parameters (e. g. STRUCT, ULINT etc.) *) 
			(* new since 3/2021 *)
			AxisEncoderMask64 	:= 5000,	(* lword *) (* IndexOffset= 16#0001_0015 *)
			AxisEncoderSubMask64,			(* lword *) (* IndexOffset= 16#0001_0108 *)
			
			{attribute 'hide'}
			AxisMasPositionDeviationAuxAxis:=32000(* lreal *)	(* IndexOffset= 16#0000_0109 *) (* added for compatibility reasons (write error AxisMasPositionDeviationAuxAxis changed to AxisMaxPositionDeviationAuxAxis) 2018-05-03 KSt *)
			);
END_TYPE

// Data types/Status and Parameter/MC_AxisStates
(* 	PLCopen axis states
	The axis states are defined in the PLCopen state diagram
*)
TYPE MC_AxisStates :
 (
	MC_AXISSTATE_UNDEFINED,
	MC_AXISSTATE_DISABLED,
	MC_AXISSTATE_STANDSTILL,
	MC_AXISSTATE_ERRORSTOP,
	MC_AXISSTATE_STOPPING,
	MC_AXISSTATE_HOMING,
	MC_AXISSTATE_DISCRETEMOTION,
	MC_AXISSTATE_CONTINOUSMOTION,
	MC_AXISSTATE_SYNCHRONIZEDMOTION
 );
END_TYPE

// Data types/Status and Parameter/ST_AxisComponents
TYPE ST_AxisComponents :
STRUCT
	EncoderIDs	: ARRAY[1..9] OF DWORD;
	ControllerIDs 	: ARRAY[1..9] OF DWORD;
	DriveIDs 		: ARRAY[1..9] OF DWORD;
END_STRUCT
END_TYPE

// Data types/Status and Parameter/ST_AxisOpModes
(* axis operation mode feedback from NcToPlc. *)
TYPE ST_AxisOpModes :
STRUCT
	PositionAreaMonitoring 	: BOOL;	(* bit 0 - OpModeDWord *)
	TargetPositionMonitoring 	: BOOL;	(* bit 1 - OpModeDWord *)
	LoopMode				: BOOL;	(* bit 2 - OpModeDWord - loop mode for two speed axes *)
	MotionMonitoring			: BOOL;	(* bit 3 - OpModeDWord *)
	PEHTimeMonitoring		: BOOL;	(* bit 4 - OpModeDWord *)
	BacklashCompensation	: BOOL;	(* bit 5 - OpModeDWord *)
	DelayedErrorReaction		: BOOL;	(* bit 6 - OpModeDWord  *)
	Modulo					: BOOL;	(* bit 7 - OpModeDWord - axis is parameterized as modulo axis *)
	SimulationAxis			: BOOL;	(* bit 8 - OpModeDWord - axis is a simulation axis - available from 2.11 R2 B2033 - 2011-05-31 KSt *)
	StopMonitoring			: BOOL;	(* bit 12 - OpModeDWord - TargetPositionMonitoring for Stop and Halt commands - available from 2.11 R3 - 2011-12-09 KSt *)
	PositionLagMonitoring		: BOOL;	(* bit 16 - OpModeDWord *)
	VelocityLagMonitoring		: BOOL;	(* bit 17 - OpModeDWord *)
	SoftLimitMinMonitoring		: BOOL;	(* bit 18 - OpModeDWord *)
	SoftLimitMaxMonitoring		: BOOL;	(* bit 19 - OpModeDWord *)
	PositionCorrection			: BOOL;	(* bit 20 - OpModeDWord *)
	AllowSlaveCommands		: BOOL;	(* bit 21 - OpModeDWord - allow motion commands on slave axes with automatic decoupling *) 	(* 2009-02-20 KSt *)
	AllowExtSetAxisCommands	: BOOL;	(* bit 22 - OpModeDWord - allow motion commands on external set point generator axes with automatic fall back to PTP mode *) 	(* 2011-10-13 KSt *)
END_STRUCT
END_TYPE

// Data types/Status and Parameter/ST_AxisParameterSet
TYPE ST_AxisParameterSet :
STRUCT
	(* AXIS: *)
	AxisId 						: DWORD;				(* 0x00000001 *) (* TC3 &&&&&&&&&&&&&&&&&&&&&&&&&&&&&&&&&&&&& *)
	nAxisType					: E_NcAxisType;			(* 0x00000003 *)
	sAxisName 					: STRING(31);			(* 0x00000002 *)
	fAxisCycleTime	 			: LREAL;				(* 0x00000004 *) (* available from Tc 2.11 R2 *)
	bEnablePositionAreaControl 	: WORD;					(* 0x0000000F *)
{attribute 'hide'}
	sReserved1					: WORD;
{attribute 'hide'}
	sReserved2					: DWORD;
	fPositionAreaControlRange 	: LREAL;				(* 0x00000010 *)
	bEnableMotionControl		: WORD;					(* 0x00000011 *)
{attribute 'hide'}
	sReserved3					: WORD;
{attribute 'hide'}
	sReserved4					: DWORD;
	fMotionControlTime 			: LREAL;				(* 0x00000012 *)
	bEnableLoop 				: WORD;					(* 0x00000013 *)
{attribute 'hide'}
	sReserved5					: WORD;
{attribute 'hide'}
	sReserved6					: DWORD;
	fLoopDistance 				: LREAL;				(* 0x00000014 *)
	bEnableTargetPosControl 	: WORD;					(* 0x00000015 *)
{attribute 'hide'}
	sReserved7					: WORD;
{attribute 'hide'}
	sReserved8					: DWORD;
	fTargetPosControlRange 		: LREAL;				(* 0x00000016 *)
	fTargetPosControlTime 		: LREAL;				(* 0x00000017 *)
	fVeloMaximum 				: LREAL;				(* 0x00000027 *)
	fRefVeloSearch				: LREAL;				(* 0x00000006 calibration velo (TO plc cam)		(17.05.11: parameter extension) *)
	fRefVeloSync				: LREAL;				(* 0x00000007 calibration velo (off plc cam)	(17.05.11: parameter extension) *)
	fVeloSlowManual				: LREAL;				(* 0x00000008 manual velocity (slow)			(17.05.11: parameter extension) *)
	fVeloFastManual				: LREAL;				(* 0x00000009 manual velocity (fast)			(17.05.11: parameter extension) *)
	fMotionControlRange 		: LREAL;				(* 0x00000028 *)
	bEnablePEHTimeControl 		: WORD;					(* 0x00000029 *)
{attribute 'hide'}
	sReserved9					: WORD;
{attribute 'hide'}
	sReserved10					: DWORD;
	fPEHControlTime 			: LREAL;				(* 0x0000002A *)
	bEnableBacklashCompensation : WORD;					(* 0x0000002B *)
{attribute 'hide'}
	sReserved11					: WORD;
{attribute 'hide'}
	sReserved12					: DWORD;
	fBacklash 					: LREAL;				(* 0x0000002C *)
	sAmsNetId 					: T_AmsNetId;			(* 0x00000031 (Wandlung von "BYTE b[6]" zum nullterminierten STRING mit 23+1 Zeichen) *)
	nPort 						: WORD;					(* 0x00000031 *)
	nChnNo 						: WORD;					(* 0x00000031 *)
{attribute 'hide'}
	sReserved13					: DWORD;
	fAcceleration 				: LREAL;				(* 0x00000101 *)
	fDeceleration 				: LREAL;				(* 0x00000102 *)
	fJerk 						: LREAL;				(* 0x00000103 *)

	(* ENCODER: *)
	nEncId 						: DWORD;				(* 0x00010001 *)
	nEncType 					: E_NcEncoderType;		(* 0x00010003 *)
	sEncName 					: STRING(31);			(* 0x00010002 *)
	fEncScaleFactorNumerator	: LREAL;				(* 0x00010023 *)
	fEncScaleFactorDenominator 	: LREAL;				(* 0x00010024 *)
	fEncScaleFactorInternal		: LREAL;				(* 0x00010006 *) (* fEncScaleFactorInternal = fEncScaleFactorNumerator / fEncScaleFactorDenominator *)
	fEncOffset 					: LREAL;				(* 0x00010007 *)
	bEncIsInverse 				: WORD;					(* 0x00010008 *)
{attribute 'hide'}
	sReserved14					: WORD;
{attribute 'hide'}
	sReserved15					: DWORD;
	fEncModuloFactor 			: LREAL;				(* 0x00010009 *)
	nEncMode 					: DWORD;				(* 0x0001000A *)
	bEncEnableSoftEndMinControl : WORD;					(* 0x0001000B *)
	bEncEnableSoftEndMaxControl : WORD;					(* 0x0001000C *)
	fEncSoftEndMin 				: LREAL;				(* 0x0001000D *)
	fEncSoftEndMax				: LREAL;				(* 0x0001000E *)
	nEncMaxIncrement 			: DWORD;				(* 0x00010015 *)
	nEncRefSoftSyncMask			: DWORD;				(* 0x00010108 *)
	bEncEnablePosCorrection 	: WORD;					(* 0x00010016 *)
{attribute 'hide'}
	sReserved16					: WORD;
	nEncReferenceSystem			: DWORD;				(* 0x00010019	(15.10.15: parameter extension) *)
	fEncPosCorrectionFilterTime : LREAL;				(* 0x00010017 *)
	(* ENCODER (incremental): *)
	bEncRefSearchInverse		: UINT;					(* 0x00010101 	(17.05.11: parameter extension) *)
	bEncRefSyncInverse			: UINT;					(* 0x00010102 	(17.05.11: parameter extension) *)
	nEncRefMode					: UDINT;				(* 0x00010107 	(17.05.11: parameter extension) *)
	fEncRefPosition				: LREAL;				(* 0x00010103 	(17.05.11: parameter extension) *)

	(* CONTROLLER: *)
	nCtrlId 					: DWORD;				(* 0x00020001 *)
	nCtrlType 					: DWORD;				(* 0x00020003 *)
	sCtrlName 					: STRING(31);			(* 0x00020002 *)
	bCtrlEnablePosDiffControl 	: WORD;					(* 0x00020010 *)
	bCtrlEnableVeloDiffControl 	: WORD;					(* 0x00020011 *)
{attribute 'hide'}
	nReserved17					: DWORD;
	fCtrlPosDiffMax				: LREAL;				(* 0x00020012 *)
	fCtrlPosDiffMaxTime 		: LREAL;				(* 0x00020013 *)
	fCtrlPosKp 					: LREAL;				(* 0x00020102 *)
	fCtrlPosTn 					: LREAL;				(* 0x00020103 *)
	fCtrlPosTv 					: LREAL;				(* 0x00020104 *)
	fCtrlPosTd 					: LREAL;				(* 0x00020105 *)
	fCtrlPosExtKp 				: LREAL;				(* 0x00020106 *)
	fCtrlPosExtVelo 			: LREAL;				(* 0x00020107 *)
	fCtrlAccKa 					: LREAL;				(* 0x00020108 *)

	(* DRIVE: *)
	nDriveId 					: DWORD;				(* 0x00030001 *)
	nDriveType 					: E_NcDriveType;		(* 0x00030003 *)
	sDriveName 					: STRING(31);			(* 0x00030002 *)
	bDriveIsInverse 			: WORD;					(* 0x00030006 *)
{attribute 'hide'}
	nReserved18					: WORD;
	nDriveControlDWord			: DWORD;				(* 0x00030010 *)
	fDriveVeloReferenz 			: LREAL;				(* 0x00030101 *)
	fDriveOutputReferenz 		: LREAL;				(* 0x00030102 *)
	fDriveOutputScalingAcc		: LREAL;				(* 0x0003000A	(15.10.15: parameter extension) *)
	fDriveOutputScalingTorque	: LREAL;				(* 0x0003000B	(15.10.15: parameter extension) *)
	fDriveInputScalingTorque	: LREAL;				(* 0x00030031	(15.10.15: parameter extension) *)
	fDriveInputFiltertimeTorque	: LREAL;				(* 0x00030032	(15.10.15: parameter extension) *)
	fDriveInputFiltertimeTorqueDerivative	: LREAL;	(* 0x00030033	(15.10.15: parameter extension) *)

	fAccelerationMax			: LREAL;				(* 0x000000F1	(15.10.15: parameter extension) *)
	fDecelerationMax			: LREAL;				(* 0x000000F2	(15.10.15: parameter extension) *)
//	fJerkMax					: LREAL;				(* 0x000000F3	(15.10.15: parameter extension) *)
	
	(* fill up *)
{attribute 'hide'}
	arrReserved : ARRAY[653..1024] OF BYTE;		(* fill up to 1024 bytes *)
END_STRUCT
END_TYPE

// Data types/Status and Parameter/ST_AxisStatus
TYPE ST_AxisStatus :
STRUCT
	UpdateTaskIndex	: 	BYTE;	(* Task-Index of the task that updated this data set *)
	UpdateCycleTime	:	LREAL;	(* task cycle time of the task which calls the status function *)
	CycleCounter		: 	UDINT;	(* PLC cycle counter when this data set updated *)
	NcCycleCounter	: 	UDINT;	(* NC cycle counter incremented after NC task updated NcToPlc data structures *)

	MotionState 		: 	MC_AxisStates; 	(* motion state in the PLCopen state diagram *)

	Error			:	BOOL;	(* StateDWord bit 31 - axis error state *)
{attribute 'displaymode':='hex'}
	ErrorID			:	UDINT;	(* axis error code *)

	(* PLCopen motion control statemachine states: *)
	ErrorStop		:	BOOL;
	Disabled			:	BOOL;
	Stopping			:	BOOL;
	StandStill		:	BOOL;
	DiscreteMotion	:	BOOL;
	ContinuousMotion	:	BOOL;	(* StateDWord bit 19 *)
	SynchronizedMotion:	BOOL;
	Homing			:	BOOL;

	(* additional status - (PLCopen definition)*)
	ConstantVelocity	:	BOOL;	(* StateDWord bit 12 *)
	Accelerating		:	BOOL;
	Decelerating		:	BOOL;

	(* Axis.NcToPlc.StateDWord *)
	Operational 		: 	BOOL;	(* StateDWord bit 0 - (was ready) *)
	ControlLoopClosed : 	BOOL;	(* StateDWord bit 20 - operational and position control active *)
	HasJob			: 	BOOL;	(* StateDWord bit 8 *)
	HasBeenStopped	: 	BOOL;	(* StateDWord bit 7 *)
	NewTargetPosition: 	BOOL;	(* StateDWord bit 17 - new target position commanded during move *)
	InPositionArea 	: 	BOOL;	(* StateDWord bit 3 *)
	InTargetPosition 	:	BOOL;	(* StateDWord bit 4 *)
	ProtectedMode	:	BOOL;	(* StateDWord bit 5 *)
	Homed			: 	BOOL;	(* StateDWord bit 1 *)
	HomingBusy		: 	BOOL;	(* StateDWord bit 11 *)
	MotionCommandsLocked 	: BOOL; (* StateDWord bit 29 - stop 'n hold *)
	SoftLimitMinExceeded		: BOOL; (* StateDWord bit 26 - reverse soft travel limit exceeded *)
	SoftLimitMaxExceeded		: BOOL; (* StateDWord bit 27 - forward soft travel limit exceeded *)

	Moving			: 	BOOL;	(* StateDWord bit 9+10 *)
	PositiveDirection	: 	BOOL;	(* StateDWord bit 9 *)
	NegativeDirection : 	BOOL;	(* StateDWord bit 10 *)
	NotMoving		:	BOOL;	(* StateDWord bit 2 *)
	Compensating	: 	BOOL;	(* StateDWord bit 13 *) (* superposition - overlayed motion *)

	ExtSetPointGenEnabled : BOOL;	(* StateDWord bit 14 *)
	PhasingActive		: BOOL;		(* StateDWord bit 15 *)
	ExternalLatchValid	: 	BOOL;	(* StateDWord bit 16 *)
	CamDataQueued	: 	BOOL;	(* StateDWord bit 22 *)
	CamTableQueued :	BOOL;	(* StateDWord bit 21 *)
	CamScalingPending : 	BOOL;	(* StateDWord bit 23 *)
	CmdBuffered 		: 	BOOL;	(* StateDWord bit 24 *)
	PTPmode 		: 	BOOL;	(* StateDWord bit 25 *)
	DriveDeviceError	: 	BOOL;	(* StateDWord bit 28 *)
	IoDataInvalid 		: 	BOOL;	(* StateDWord bit 30 *)
	ErrorPropagationDelayed	: BOOL;	(* StateDWord bit 6 *)
	DriveLimitActive			: BOOL;(* StateDWord bit 18 - 20181213 Fap*)

	(* Axis.NcToPlc.CoupleState *)
	Coupled			: 	BOOL;

	(* axis operation mode feedback from NcToPlc *)
	OpMode			: 	ST_AxisOpModes;
	NcApplicationRequest : BOOL; 		(* OpModeDWord bit 23 *)
END_STRUCT
END_TYPE

// Data types/Status and Parameter/ST_DriveAddress
TYPE ST_DriveAddress :
STRUCT
	NetID					: T_AmsNetId;		(* AMS NetID of the hardware drive as a string *)
	NetIdBytes				: T_AmsNetIdArr;	(* AMS NetID of the hardware drive as a byte array (same information as NetID) *)
	SlaveAddress			: T_AmsPort;		(* slave address of the hardware drive connected to a bus master *)
	Channel					: BYTE;				(* channel number of the hardware drive *)
	(* new since 2013-04-04 KSt - just available with versions after this date, otherwise zero *)
	NcDriveId 				: DWORD;			(* ID [1..255] of the NC software drive of an axis *)
	NcDriveIndex 			: DWORD;			(* index [0..9] of the NC software drive of an axis *)
	NcDriveType 			: E_NcDriveType;	(* type enumeration of the NC software drive of an axis *)
	NcEncoderId 			: DWORD;			(* ID [1..255] of the NC software encoder of an axis *)
	NcEncoderIndex 			: DWORD;			(* index [0..9] of the NC software encoder of an axis *)
	NcEncoderType 			: E_NcEncoderType;	(* type enumeration of the NC encoder drive of an axis *)
	NcAxisId 				: DWORD;			(* ID [1..255] of the NC axis *)
	NcAxisType 				: E_NcAxisType;		(* type enumeration of the NC axis *)
	(* new since 2016-04-11 FAP - just available with versions after this date, otherwise zero *)
	{attribute 'conditionalshow'}
	TcSoftDriveObjectId		: OTCID;	
	TcDriveObjectId			: OTCID;
	TcEncoderObjectId		: OTCID;
	TcAxisObjectId			: OTCID;
END_STRUCT
END_TYPE

// Data types/Status and Parameter/ST_McOutputs
TYPE ST_McOutputs :
STRUCT
	Done				:	BOOL;
	Busy 				: 	BOOL;
	Active	 			: 	BOOL;
	CommandAborted		:	BOOL;
	Error				:	BOOL;
{attribute 'displaymode':='hex'}	
	ErrorID				:	UDINT;
END_STRUCT
END_TYPE

// Data types/Status and Parameter/ST_NcApplicationRequest
TYPE ST_NcApplicationRequest :
STRUCT
	(* APPLICATION REQUEST DATA: *)
	bApplRequestBit 				: UINT;		(* application request bit [0/1] *)
	nApplRequestType 				: UINT;		(* application request TYPE/ID *)
	nApplRequestCounter				: UDINT;	(* continuous actual command number *)
	nApplRequestVersion 			: UDINT;	(* application command version (structure version), 01.04.10: 'V0' *)
	
	(**)
{attribute 'hide'}
	nReserved1 					: ARRAY[13..1024] OF BYTE;		(* fill up to 1024 bytes *)
END_STRUCT
END_TYPE

// Data types/Status and Parameter/ST_PowerOptions
TYPE ST_PowerOptions :
STRUCT
	; 	(* empty so far xxx *)
END_STRUCT
END_TYPE

// Data types/Status and Parameter/ST_SetEncoderScalingOptions
TYPE ST_SetEncoderScalingOptions :
STRUCT
	SelectEncoderIndex 	: BOOL;	(* selects an encoder with index 0..n explicitly if enabled - selction by EncoderIndex below *)
	EncoderIndex 		: UINT;	(* encoder with index 0..n, 0 is first encoder - valid only if SelectEncoderIndex=TRUE *)
END_STRUCT
END_TYPE

// Data types/Status and Parameter/ST_SetPositionOptions
TYPE ST_SetPositionOptions :
STRUCT
	ClearPositionLag 		: BOOL;	(* set actual and set position to same value and clear the position lag *)
	SelectEncoderIndex 	: BOOL;	(* selects an encoder with index 0..n explicitly if enabled - selction by EncoderIndex below *)
	EncoderIndex 		: UINT;	(* encoder with index 0..n, 0 is first encoder - valid only if SelectEncoderIndex=TRUE *)
END_STRUCT
END_TYPE

// Data types/Status and Parameter/ST_TableCharacValues
{attribute 'conditionalshow'}
TYPE ST_TableCharacValues :
STRUCT
    (* Master Velocity*)
	fMasterVeloNom	: LREAL;    (* 1.  master nominal velocity (normed: => 1.0) *)

	(* characteristic slave data *)
	(*===========================*)

   (* Start of cam table *)
	fMasterPosStart	: LREAL;	(* 2.  master start position *)
	fSlavePosStart	: LREAL;	(* 3.  slave start position *)
	fSlaveVeloStart	: LREAL;	(* 4.  slave start velocity *)
	fSlaveAccStart	: LREAL;	(* 5.  slave start acceleration *)
	fSlaveJerkStart	: LREAL;	(* 6.  slave start jerk *)

	(* End of cam table*)
	fMasterPosEnd	: LREAL;	(* 7.  master end position *)
	fSlavePosEnd	: LREAL;	(* 8.  slave end position *)
	fSlaveVeloEnd	: LREAL;	(* 9.  slave end velocity *)
	fSlaveAccEnd	: LREAL;	(* 10. slave end acceleration *)
	fSlaveJerkEnd	: LREAL;	(* 11. slave end jerk *)

	(* minimum slave position *)
	fMPosAtSPosMin	: LREAL;	(* 12. master position AT slave minimum position *)
	fSlavePosMin	: LREAL;	(* 13. slave minimum position *)

	(* minimum Slave velocity *)
	fMPosAtSVeloMin	: LREAL;	(* 14. master position AT slave minimum velocity *)
	fSlaveVeloMin	: LREAL;	(* 15. slave minimum velocity *)

	(* minimum slave acceleration *)
	fMPosAtSAccMin	: LREAL;	(* 16. master position AT slave minimum acceleration *)
	fSlaveAccMin	: LREAL;	(* 17. slave minimum acceleration *)
	fSVeloAtSAccMin	: LREAL;	(* 18. slave velocity AT slave minimum acceleration *)

	(* minimum slave jerk and dynamic momentum *)
	fSlaveJerkMin	: LREAL;	(* 19. slave minimum jerk *)
	fSlaveDynMomMin	: LREAL;	(* 20. slave minimum dynamic momentum (NOT SUPPORTED YET !) *)

	(* maximum slave position *)
	fMPosAtSPosMax	: LREAL;	(* 21. master position AT slave maximum position *)
	fSlavePosMax	: LREAL;	(* 22. slave maximum position *)

	(* maximum Slave velocity *)
	fMPosAtSVeloMax	: LREAL;	(* 23. master position AT slave maximum velocity *)
	fSlaveVeloMax	: LREAL;	(* 24. slave maximum velocity *)

	(* maximum slave acceleration *)
	fMPosAtSAccMax	: LREAL;	(* 25. master position AT slave maximum acceleration *)
	fSlaveAccMax	: LREAL;	(* 26. slave maximum acceleration *)
	fSVeloAtSAccMax	: LREAL;	(* 27. slave velocity AT slave maximum acceleration *)

	(* maximum Slave slave jerk and dynamic momentum *)
	fSlaveJerkMax	: LREAL;	(* 28. slave maximum jerk *)
	fSlaveDynMomMax	: LREAL;	(* 29. slave maximum dynamic momentum (NOT SUPPORTED YET !) *)

	(* mean and effective values *)
	fSlaveVeloMean	: LREAL;	(* 30. slave mean absolute velocity (NOT SUPPORTED YET !) *)
	fSlaveAccEff	: LREAL;	(* 31. slave effective acceleration (NOT SUPPORTED YET !) *)

	(* reserved space for future extension *)
{attribute 'hide'}
	reserved 		: ARRAY[32..47] OF LREAL;

	(* organization structure of the cam table *)
	CamTableID 			: UDINT;
	NumberOfRows		: UDINT;	(* number of cam table entries, e. g. number of points *)
	NumberOfColumns	: UDINT;	(* number of table columns, typically 1 or 2 *)
	TableType			: INT;
	Periodic				: BOOL;

{attribute 'hide'}
	reserved2 		: ARRAY[1..121] OF BYTE;
END_STRUCT
END_TYPE

// Data types/Stepper/E_DestallDetectMode
TYPE E_DestallDetectMode :
	(
		PwStDetectMode_None := 0,		(* do not detect stall situations *)
		PwStDetectMode_Encoderless,		(* use status signals of KL2531/KL2541 for stall detection *)
		PwStDetectMode_Lagging			(* use encoder signals for stall detection *)
	);
END_TYPE

// Data types/Stepper/E_DestallMode
TYPE E_DestallMode :
	(
		PwStMode_None := 0,			(* do not respond to stall situations *)
		PwStMode_SetError,			(* in stall situations place axis in fault state *)
		PwStMode_SetErrNonRef,		(* in stall situations place axis in nonreferenced state *)
		PwStMode_UseOverride			(* use override to catch the axis and recover from stall situations *)
	);
END_TYPE

// Data types/Stepper/ST_PowerStepperStruct
TYPE ST_PowerStepperStruct :
STRUCT
	DestallDetectMode	:	E_DestallDetectMode;
	DestallMode			:	E_DestallMode;
	DestallEnable		:	BOOL;
	StatusMonEnable		:	BOOL;

	Retries				:	INT;
	Timeout				:	TIME;
END_STRUCT
END_TYPE

// Data types/Superposition/E_SuperpositionAbortOption
TYPE E_SuperpositionAbortOption :
 (
 	SUPERPOSITIONOPTION_ABORTATSTANDSTILL := 0,	(* aborts the superposition when the subordinated motion profile velocity is zero - standard of  MC_MoveSuperimposed (TcMC version 1) *)
 	SUPERPOSITIONOPTION_RESUMEAFTERSTANDSTILL,	(* resumes the superposition after a temporary standstill of the subordinated motion profile *)
 	SUPERPOSITIONOPTION_RESUMEAFTERMOTIONSTOP	(* resumes the superposition after any stop and restart of the subordinated motion profile - ResumeAfterMotionStop includes ResumeAfterStandstill *)
 ) UINT;
END_TYPE

// Data types/Superposition/E_SuperpositionMode
TYPE E_SuperpositionMode :
 (
 	SUPERPOSITIONMODE_VELOREDUCTION_ADDITIVEMOTION := 1,	(* standard type of  MC_MoveSuperimposed (TcMC version 1) *)
 	SUPERPOSITIONMODE_VELOREDUCTION_LIMITEDMOTION,
 	SUPERPOSITIONMODE_LENGTHREDUCTION_ADDITIVEMOTION,
 	SUPERPOSITIONMODE_LENGTHREDUCTION_LIMITEDMOTION,
 	SUPERPOSITIONMODE_ACCREDUCTION_ADDITIVEMOTION,			(* new 2009-05 *)
 	SUPERPOSITIONMODE_ACCREDUCTION_LIMITEDMOTION			(* new 2009-05 *)
 ) UINT;
END_TYPE

// Data types/Superposition/ST_SuperpositionOptions
TYPE ST_SuperpositionOptions :
STRUCT
	AbortOption : E_SuperpositionAbortOption;
END_STRUCT
END_TYPE

// Data types/Torque Control/ST_TorqueControlOptions
TYPE ST_TorqueControlOptions :
STRUCT
	EnableManualTorqueStartValue: BOOL;

	ManualTorqueStartValue		: LREAL;
END_STRUCT
END_TYPE

// Data types/Touch Probe/E_SignalEdge
(* signal edge used with MC_TouchProbe *)
TYPE E_SignalEdge :
 (
	RisingEdge,
	FallingEdge
 ) UINT;
END_TYPE

